(* write scene if necessary *)
IF swrite THEN
	status := 176;		(* write scene *)
	sx[x,0] := pi;
	sx[x,1] := ai;
	IF enable THEN sx[x,2] := 1; ELSE sx[x,2] := 0; END_IF; (* if sx[x,2] = 0 the scene is disabled *)
END_IF;


(* revision history
hm	24. oct 2007	rev 1.0
	original release

hm		29.1.2008	rev 1.1
	replaced shr/shl with and for better performance
*)
END_FUNCTION_BLOCK

(* POU BLIND_SECURITY, ST *)
FUNCTION_BLOCK BLIND_SECURITY
VAR_INPUT
	UP, DN : BOOL;
	S_IN : BYTE;
	pi, ai : BYTE;
	FIRE : BOOL;
	Wind : BOOL;
	Alarm : BOOL;
	Door : BOOL;
	Rain : BOOL;
END_VAR
VAR_INPUT CONSTANT
	Alarm_UP : BOOL := TRUE;
	WIND_UP :BOOL := TRUE;
	RAIN_UP : BOOL := FALSE;
END_VAR
VAR_OUTPUT
	QU, QD : BOOL;
	status : BYTE;
	po, ao : BYTE;
END_VAR
VAR
END_VAR

(*
version 1.2	12. feb 2008
programmer 	hugo
tested by		tobias


*)
IF Fire THEN
	QU := TRUE;
	QD := FALSE;
	status := 111;
ELSIF Wind THEN
	QU := Wind_up;
	QD := NOT wind_up;
	status := 112;
ELSIF alarm THEN
	QU := Alarm_up;
	QD := NOT Alarm_up;
	status := 113;
ELSIF Door THEN
	QU := TRUE;
	QD := FALSE;
	status := 114;
ELSIF Rain AND NOT (up XOR dn) THEN
	QU := rain_up;
	QD := NOT rain_up;
	status := 115;
ELSE
	QU := UP;
	QD := DN;
	status := S_IN;
	po := pi;
	ao := ai;
END_IF;


(* revision history
hm	29. sep 2007	rev 1.0
	original release

hm	6. oct 2007		rev 1.1
	added pos and angle inputs and outputs
	manual will override rain position
	alarm position can now be configured

hm		12. feb. 2008	rev 1.2
	added config variables rain_up and wind_up
	position for rain and wind is now configurable
*)
END_FUNCTION_BLOCK

(* POU BLIND_SHADE, ST *)
FUNCTION_BLOCK BLIND_SHADE
VAR_INPUT
	UP, DN : BOOL;
	S_IN : BYTE;
	pi, ai : BYTE;
	enable : BOOL;
	sun : BOOL;
	dtin : DT;
	sunrise, sunset : TOD;
	sun_hor, sun_ver : REAL;
END_VAR
VAR_INPUT CONSTANT
	sunrise_offset : TIME := T#1h;
	sunset_preset : TIME := T#1h;
	direction : REAL := 180;
	angle_offset : REAL := 80;
	slat_width : REAL := 80;
	Slat_spacing : REAL := 60;
	Shade_delay : TIME := T#60s;
END_VAR
VAR_OUTPUT
	QU, QD : BOOL;
	status : BYTE;
	po, ao : BYTE;
END_VAR
VAR
	angle: REAL;
	sun_delay : TOF;
END_VAR

(*
version 1.2	24 nov 2007
programmer 	hugo
tested by		tobias


*)
(* the input sun is sent through tof which will delay the shade for the time shade_delay *)
sun_delay(IN := sun, PT := shade_delay);

IF UP AND DN AND enable AND sun_delay.Q AND sun_hor > direction - angle_offset AND sun_hor < direction + angle_offset AND
	DT_TO_TOD(dtin) > sunrise + sunrise_offset AND DT_TO_TOD(dtin) < sunset - sunset_preset THEN
	status := 151;
	QU := UP;
	QD := DN;
	(* position is fully down *)
	po := 0;
	(* shading is active now calculate the slat angle *)
	(* calculate the max angle for the blind *)
	angle := DEG(ATAN(slat_spacing / slat_width));
	(* check if sun angle is between 0 and max angle *)
	IF sun_ver > 0 AND sun_ver < angle THEN
		angle := sun_ver + DEG(ACOS(COS(RAD(sun_ver))*slat_spacing / Slat_width));
		ao := INT_TO_BYTE(LIMIT(0,TRUNC(angle * 255 / 90), 255));
	ELSE
		ao := 255;
	END_IF;
ELSE
	QU := UP;
	QD := DN;
	po := pi;
	ao := ai;
	status := S_IN;
END_IF;

(* revision history
hm	15 oct. 2007	rev 1.0
	original version

hm	19. oct 2007	rev 1.1
	manual mode was not detected because outputs were checked and not inputs UP and DN

hm	24. nov 2007	rev 1.2
	added shade_delay to avoid constant up and down if sun is out parcially
*)
END_FUNCTION_BLOCK

(* POU DEG, ST *)
FUNCTION DEG : REAL
VAR_INPUT
	rad : REAL;
END_VAR
VAR
END_VAR
VAR
END_VAR

(*
version 1.1	16 oct 2007
programmer 	hugo
tested by		tobias

this function converts degrees into Radiant
execution time on wago 750 - 841 =  10  us
*)
deg := modR(57.29577951308232 * Rad, 360);

(* revision history
hm	4. aug 2006		rev 1.0
	original version

hm 	16. oct 2007	rev 1.1
	added modr statement which prohibits deg to become bigger than 360

*)
END_FUNCTION

(* POU RAD, ST *)
FUNCTION RAD : REAL
VAR_INPUT
	deg : REAL;
END_VAR
VAR
END_VAR

(*
version 1.0	4 aug 2006
programmer 	hugo
tested by	tobias

this function converts Radiant to degrees

*)
Rad := modR(0.0174532925199433 * deg,PI2);

(* revision history
hm	4. aug 2006
	original version

hm 	16. oct 2007
	added modr statement which prohibits rad to become bigger than 2PI

*)
END_FUNCTION

(* POU MODR, ST *)
FUNCTION MODR : REAL
VAR_INPUT
	in : REAL;
	divi : REAL;
END_VAR

VAR
END_VAR

(*
version 1.3	4. apr. 2008
programmer 	hugo
tested by	tobias

this is a modulo funtion for real numbers
modr(5.5,2.5) = 0.5

*)
IF divi = 0 THEN
	MODR := 0;
ELSE
	MODR := in - DINT_TO_REAL(D_TRUNC(in / divi)) * divi;
END_IF;

(* revision history

hm	4. aug.2006		rev 1.0

hm	28. jan.2007	rev 1.1
	modr(x,0) will deliver the result 0

hm	21. mar 2008	rev 1.2
	use D_trunc for compatibility reasons

hm	4. apr. 2008	rev 1.3
	added type conversion to avoid warnings under codesys 3.0

*)
END_FUNCTION

(* POU BOILER, ST *)
FUNCTION_BLOCK BOILER
VAR_INPUT
	T_upper : REAL;
	T_lower : REAL;
	Pressure : BOOL := TRUE;
	enable : BOOL := TRUE;
	Req_1 : BOOL;
	Req_2 : BOOL;
	Boost : BOOL;
END_VAR
VAR_INPUT CONSTANT
	t_upper_min : REAL := 50;
	t_upper_max : REAL := 60;
	T_lower_enable : BOOL;
	T_lower_max : REAL := 60;
	T_request_1 : REAL := 70;
	T_request_2 : REAL := 50;
	T_request_hys : REAL := 5;
	T_protect_high : REAL := 80;
	T_protect_low : REAL := 10;
END_VAR
VAR_OUTPUT
	Heat : BOOL;
	error : BOOL;
	status : BYTE;
END_VAR
VAR
	edge: BOOL;
	boost_mode: BOOL;
	flag_0 : BOOL;
	flag_1: BOOL;
	flag_2: BOOL;
END_VAR

(*
version 1.0	27 feb 2007
programmer 	hugo
tested by		tobias

this function block controls a hot water boiler. The Boiler can be equipped with two temperature sensors on top and bottom of the tank, T_LOWER_ENABLE must be set to True in this case.
alternatively can BOILER be configured for one (TOP) temperature sensor only (T_LOWER_ENABLE set to False).
A Pressure sensor is used to detect fresh water pressure and disable all heating if there is no water pressure. This input is dset to True by default, so if it is not used it can simply be left open.
A enable input enables the hot water heating while it is set to True. alternatively can a Ture on Req_1 or Req_2 start the heating to predefined temperatures during setup.
A low to high edge on the boost input will start heating imediately until T_upper_max is reached, it can be used to generate extra hot water when needed.

*)
(* read sensors and check for valid data *)
IF t_upper > t_protect_high THEN
	status := 1;
	heat := FALSE;
	error := TRUE;
ELSIF t_upper < t_protect_low THEN
	status := 2;
	heat := TRUE;
	error := TRUE;
ELSIF t_lower > T_protect_high AND t_lower_enable THEN
	status := 3;
	heat := FALSE;
	error := TRUE;
ELSIF t_lower < t_protect_low AND t_lower_enable THEN
	status := 4;
	heat := TRUE;
	error := TRUE;
ELSIF NOT pressure THEN
	status := 5;
	heat := FALSE;
	error := TRUE;
ELSIF req_1 OR req_2 OR enable OR boost THEN
	error := FALSE;

	(* determine if heat needs to be turned on *)
	IF boost AND NOT edge AND t_upper < t_upper_max THEN
		status := 101;
		heat := TRUE;
		boost_mode := TRUE;
	ELSIF enable AND t_upper < T_upper_min THEN
		status := 102;
		heat := TRUE;
	ELSIF req_1 AND t_upper < T_request_1 THEN
		status := 103;
		heat := TRUE;
	ELSIF req_2 AND t_upper < t_request_2 THEN
		status := 104;
		heat := TRUE;
	END_IF;

	(* determine the shut off temperature *)
	IF heat THEN
		IF (enable OR boost_mode) THEN
			flag_0 := TRUE;
			IF T_lower_enable AND T_lower > T_lower_max THEN
				flag_0 := FALSE;
				boost_mode := FALSE;
			ELSIF NOT T_lower_enable AND T_upper > T_upper_max THEN
				flag_0 := FALSE;
				boost_mode := FALSE;
			END_IF;
		ELSE
			flag_0 := FALSE;
		END_IF;
		IF req_1 AND T_upper > T_request_1 + T_request_hys THEN flag_1 := FALSE; ELSE flag_1 := req_1; END_IF;
		IF req_2 AND T_upper > T_request_2 + T_request_hys THEN flag_2 := FALSE; ELSE flag_2 := req_2; END_IF;

		(* shut off heat if no longer needed *)
		heat := flag_0 OR flag_1 OR flag_2;
		IF heat = FALSE THEN status := 100; END_IF;
	END_IF;
ELSE
	status := 100;
	heat := FALSE;
	error := FALSE;
END_IF;
edge := boost;
END_FUNCTION_BLOCK

(* POU PRESSURE, ST *)
FUNCTION_BLOCK PRESSURE
VAR_INPUT
	mws : REAL;
	torr : REAL;
	att : REAL;
	atm : REAL;
	pa : REAL;
	bar : REAL;
END_VAR
VAR_OUTPUT
	Ymws : REAL;
	Ytorr : REAL;
	Yatt : REAL;
	Yatm : REAL;
	Ypa : REAL;
	Ybar : REAL;
END_VAR
VAR
END_VAR

(*
version 1.0	27 mar 2007
programmer 	hugo
tested by		oscat

this function converts different pressure units
any unused input can simply be left open.
different inputs connected at the same time will be added up.
*)
Ybar := bar +
		pa / 100000 +
		0.980665 * att +
		1.01325 * atm +
		0.001333224 * torr +
		0.0980665 * mws;
Ymws := ybar / 0.0980665;
Ytorr := ybar / 0.001333224;
Yatt := ybar / 0.980665;
yatm := ybar / 1.01325;
Ypa := ybar * 100000;


(*
Druck, Pascal Pa 1 Pa = 1 N/m2 = 1 kg/(s2 �E m) . 0,75 �E 10.2 mmHg
mechanische 1 MPa = 1 N/mm2 . fur Festigkeitsangaben
Spannung Bar bar 1 bar = 105 Pa = 103 mbar = 105 kg/(s2 �E m)
Millimeter- mmHg 1 mmHg = 133,322 Pa = 1,333 22 mbar
Quecksilbersaule . nur in Heilkunde zulassig
physik. Atmosphare atm 1 atm = 1,013 25 bar
techn. Atmosphare at 1 at = 1 kp/cm2 = 0,980665 bar
Torr Torr 1 Torr = (101325/760) Pa = 1,333224 mbar
Meter-Wassersaule mWS 1 mWS = 9806,65 Pa = 98,0665 mbar
psi lbf/in2 1 lbf/in2 = 68,947 57 mbar = 6894,757 Pa

*)
END_FUNCTION_BLOCK

(* POU BUFFER_SEARCH, ST *)
FUNCTION BUFFER_SEARCH : INT
VAR_INPUT
	pt : POINTER TO ARRAY[0..32767] OF BYTE;
	size : UINT;
	str : STRING(STRING_LENGTH);
	pos : INT;
	ign : BYTE;
END_VAR
VAR
	ps : POINTER TO ARRAY[0..255] OF BYTE;
	i: INT;
	end: INT;
	k: INT;
	lx: INT;
END_VAR


(*
version 1.2	13. may. 2008
programmer 	hugo
tested by		tobias

this function will search for a string STR in an array of byte starting at position pos.
the function needs to be called:	buffer_search(adr("array"),sizeof("array"), STR, POS, IGN);
because this function works with pointers its very time efficient and it needs no extra memory.
The function returns the position of the first character of the string in the array if found.
a 0 is returned if the string is not found in the array.
The parameter IGN specifies a wildcard character in the search string.

*)
ps := ADR(str);
lx := LEN(str);
end := UINT_TO_INT(size) - lx;
lx := lx - 1;
FOR i := pos TO end DO
	FOR k := 0 TO lx DO
		IF (ps^[k] <> ign) AND (ps^[k] <> pt^[i+k]) THEN EXIT; END_IF;
	END_FOR;
	IF k > lx THEN
		BUFFER_SEARCH := i;
		RETURN;
	END_IF;
END_FOR;
BUFFER_SEARCH := 0;


(* revision History

hm 5. mar. 2008	rev 1.0
	original version

hm	16. mar. 2008	rev 1.1
	chaged type of input size to uint

hm	13. may. 2008	rev 1.2
	changed type of pointer to array[1..32767]
	changed size of string to STRING_LENGTH
*)
END_FUNCTION

(* POU BUFFER_TO_STRING, ST *)
FUNCTION BUFFER_TO_STRING : STRING(STRING_LENGTH)
VAR_INPUT
	pt : POINTER TO ARRAY[0..32767] OF BYTE;
	size : UINT;
	start : UINT;
	stop : UINT;
END_VAR
VAR
	ps : POINTER TO BYTE;
	i : INT;
END_VAR


(*
version 1.3	12. jun. 2008
programmer 	hugo
tested by		tobias

this function will retrieve a string from an array of byte starting at position start and stop at position stop.
the function needs to be called:	buffer_TO_String(adr("array"),sizeof("array"), start, stop);
because this function works with pointers its very time efficient and it needs no extra memory.

*)
ps := ADR(BUFFER_TO_STRING);
start :=MIN(start, size);
stop := MIN(stop, size);
(* check for maximum string_length *)
IF UINT_TO_INT(stop - start + 1) >= STRING_LENGTH THEN
	stop := start + INT_TO_UINT(string_length) - 1;
END_IF;

FOR i := UINT_TO_INT(start) TO UINT_TO_INT(stop) DO
	ps^ := pt^[i];
	ps := ps + 1;
END_FOR;

(* terminate the string *)
ps^ := 0;

(* revision History
hm 	5. mar. 2008	rev 1.0
	original version

hm	16. mar. 2008	rev 1.1
	changed type of input size to uint

hm	13. may. 2008	rev 1.2
	changed type of pointer to array[0..32767]
	changed size of string to STRING_LENGTH

hm	12. jun. 2008	rev 1.3
	check for pointer overrun
	change input start and stop to uint
	added type conversions to avoid warnings under codesys 3.0
*)
END_FUNCTION

(* POU BURNER, ST *)
FUNCTION_BLOCK BURNER
VAR_INPUT
	in : BOOL;
	stage2 : BOOL;
	over_temp : BOOL;
	oil_temp : BOOL := TRUE;
	Flame : BOOL;
	rst : BOOL;
	rst_timer : BOOL;
END_VAR
VAR_INPUT CONSTANT
	pre_heat_time : TIME := t#5s;
	pre_vent_time : TIME := t#15s;
	pre_ignite_time : TIME := t#5s;
	post_ignite_time : TIME := t#25s;
	stage2_delay : TIME := t#10s;
	safety_time : TIME := t#5s;
	lockout_time : TIME := t#10s;
	multiple_ignition : BOOL := TRUE;
	KW1 : REAL;
	KW2 : REAL;
END_VAR
VAR_OUTPUT
	motor : BOOL;
	coil1 : BOOL;
	coil2 : BOOL;
	pre_heat: BOOL;
	ignite : BOOL;
	runtime1 : REAL;
	runtime2 : REAL;
	KWh : REAL;
	cycles : REAL;
	status : BYTE;
	fail : BOOL;
END_VAR
VAR
	state : BYTE;
	last : TIME;
	tx: TIME;
	last_change: TIME;
	timer1 : ontime;
	timer2 : ontime;
	oil_temp_last: BOOL;
END_VAR

(*
version 1.5	15 sep 2007
programmer 	oscat
tested by		tobias

burner ist eine Oel-Brenner_steuerung fuer nichtmodulierende Oelbrenner
die steuerung kann ueber setup werte programmiert werden und entsprechenden brennern angepasst werden.
die vorheizzeit ist die zeit die eine oelvorwaermung aufgeheizt wird bevor der motor gestartet wird.
der eingang oil_temp gibt an ob die oil_temp erreicht wurde, er ist default auf true und kann auch offen gelassen werden.
die vorbelueftungszeit ist die zeit die der luefter laeuft bevor die oelzufuhr freigegeben wird.
die vorzuendzeit iust diejenige zeit die die zuendung vor offnen des oelventiel gestartet wird.
nachzuendzeit ist die zeit die nach entzuendung der flamme noch gezuendet wird.
die sicherheitszeit ist die zeit nach der die oelzufuhr gesperrt wird wenn keine flamme entsteht.
nach ablauf der sicherheitszeit wird ein fehler flag gesetzt und kann erst nach der sperrzeit wieder durch einen reset geloescht werden.
waehrend der sperrzeit ist keine weitere zuendung oder einschalten moeglich.
das flag mehrfachzuendung gibt an ob eine erloschene flamme in betrieb automatisch wieder gezuendet werden soll.
der flammwaechster liegt auf eingang flamme, ein uebertemperaturschutz auf dem eingang over_temp
der betriebsstundenzaehler gibt die brennerstunden in stunden als real ausgabewer an.
der ausgang motor steuert den luefter / pumpenmotor, oil_ventil schaltet das oil ventil und zuendung schaltet die zuendung ein.

if output fail > 0 an error happened and the output has an error code:
0 :	no error
1 :	pre heating time expired and oil temp input is not true
2 :	flame monitor is active during preheating time
3 :	flame monitor active during pre_ventilation_time
4 :	no ignoition during safety time
5 :	no flame during operation
9 :	overtemp input is true

*)
(* read system time *)
tx := DWORD_TO_TIME(T_PLC_MS());

(* check rst input and overtemp *)
IF rst OR over_temp OR state = 0 THEN
	IF status > 0 AND tx - last_change >= lockout_time AND rst THEN
		status := 110;
		fail := FALSE;
		state := 1;
	ELSE
		(* normaler reset *)
		motor := FALSE;
		coil1 := FALSE;
		coil2 := FALSE;
		ignite := FALSE;
		pre_heat := FALSE;
		IF over_temp THEN
			status := 9;
			fail := TRUE;
		END_IF;
		last_change := tx;
		last := tx;
		state := 1;
	END_IF;
END_IF;

(* check for timer rst and rst timer if true *)
IF rst_timer THEN
	timer1( rst := TRUE);
	timer1.rst := FALSE;
	timer2(rst := TRUE);
	timer2.rst := FALSE;
END_IF;

(* quit here if an error is present *)
IF (status > 0 AND status < 100) OR rst THEN RETURN; END_IF;

(* start sequence *)
CASE state OF

1:	(* in signal starts oil pre heating *)
	IF in AND flame THEN
		state := 7;
		pre_heat := FALSE;
		status := 2;
		last_change := tx;
	ELSIF in THEN
		pre_heat := TRUE;
		state := 2;
		last_change := tx;
	END_IF;

2:	(* after pre_heating time start motor *)
	IF (tx- last_change >= pre_heat_time AND oil_temp) OR (oil_temp AND NOT oil_temp_last) THEN
		motor := TRUE;
		state := 3;
		last_change := tx;
	(* pre_heat_time ist abgelaufen und oil_temp ist nicht aktiv *)
	ELSIF tx - last_change >= pre_heat_time AND NOT oil_temp THEN
		state := 7;
		pre_heat := FALSE;
		status := 1;
		last_change := tx;
	(* flame monitor cannot be active at this time *)
	ELSIF flame THEN
		state := 7;
		pre_heat := FALSE;
		status := 2;
		last_change := tx;
	END_IF;

3:	(* abwarten bis zündung eingeschaltet werden kann *)
	IF tx - last_change >= pre_vent_time - pre_ignite_time THEN
		ignite := TRUE;
		state := 4;
		last_change := tx;
	(* flame monitor cannot be active at this time *)
	ELSIF flame THEN
		state := 7;
		pre_heat := FALSE;
		motor := FALSE;
		status := 3;
		last_change := tx;
	END_IF;

4:	(* warten bis oelzufuhr geoeffnet werden darf *)
	IF tx - last_change >= pre_ignite_time THEN
		coil1 := TRUE;
		state := 5;
		last_change := tx;
	END_IF;

5:	(* warten auf flammwaechter und falls noetig abschalten *)
	IF tx - last_change >= safety_time OR flame THEN
		IF NOT flame THEN
			(* notabschaltung da flammwaechster nicht angesprochen hat *)
			state := 7;
			motor := FALSE;
			coil1 := FALSE;
			pre_heat := FALSE;
			ignite := FALSE;
			status := 4;
			last_change := tx;
		ELSE
			state := 6;
			last_change := tx;
		END_IF;
	END_IF;

6:	(* brenner läuft, flammueberwachung und nach ablauf der nachigniteszeit ignite abschalten *)
	IF NOT flame AND NOT multiple_ignition THEN
		(* notabschaltung da flammwaechster keine flamme meldet *)
		state := 7;
		motor := FALSE;
		coil1 := FALSE;
		coil2 := FALSE;
		pre_heat := FALSE;
		ignite := FALSE;
		status := 5;
		last_change := tx;
	ELSIF NOT flame AND multiple_ignition THEN
		ignite := TRUE;
		state := 5;
		coil2 := FALSE;
		last_change := tx;
	ELSE
		IF tx - last_change >= post_ignite_time THEN
			(* post_ignite_time abgelaufen, ignite abschalten *)
			ignite := FALSE;
		END_IF;
		IF tx - last_change >= stage2_delay AND stage2 THEN
			coil2 := TRUE;
		ELSE
			coil2 := FALSE;
		END_IF;
	END_IF;
END_CASE;

(* abschaltung wenn kein eingangssignal *)
IF NOT in THEN
	state := 1;
	motor := FALSE;
	coil1 := FALSE;
	coil2 := FALSE;
	ignite := FALSE;
	pre_heat := FALSE;
	last_change := tx;
END_IF;

(* runtimezähler *)
timer1(in := flame AND in AND motor AND coil1 AND NOT coil2);
timer2(in := flame AND in AND motor AND coil1 AND coil2);
runtime1 := timer1.ontime;
runtime2 := timer2.ontime;
cycles := timer1.cycles;
KWH := runtime1 * KW1 + runtime2 * KW2;

(* zeit fuer naechsten aufruf merken *)
last := tx;

(* set fail output IF ERROR and Status  if normal operation *)

IF status > 0 AND status < 100 THEN
	fail := TRUE;
ELSE
	fail := FALSE;
	IF NOT in THEN
		status := 110;
	ELSIF flame AND in AND motor AND coil2 AND coil1 THEN
		status := 113;
	ELSIF flame AND in AND motor AND coil1 THEN
		status := 112;
	ELSE
		status := 111;
	END_IF;
END_IF;


(*
31.12.2006	hm		rev 1.1
	added pre_heat timing and output
	flame monitor before ignition will generate error on status output
	added output for KWh

31.12.2006	hm		rev 1.2
	added oil_temp_input

31.12.2006	hm		rev 1.3
	changed status output to be byte instead of bool

22.1.2007		hm		rev 1.4
	renamed fail output to status
	added output cycles
	corrected an error while pre_heat would be on when an error was present
	added coil2 output and stage2 input

15.9.2007		hm		rev 1.5
	replaced Time() with T_PLC_MS for compatibility and performance reasons

*)
END_FUNCTION_BLOCK

(* POU BYTE_OF_BIT, ST *)
FUNCTION BYTE_OF_BIT : BYTE
VAR_INPUT
	B0:BOOL;
	B1:BOOL;
	B2:BOOL;
	B3:BOOL;
	B4:BOOL;
	B5:BOOL;
	B6:BOOL;
	B7:BOOL;
END_VAR
VAR
END_VAR

(*
version 1.1	 18. feb 2006
programmer 	hugo
tested by		tobias

this function creates a byte from 8 individual bits

*)
Byte_of_bit := SHL(SHL(SHL(SHL(SHL(SHL(SHL(BOOL_TO_BYTE(B7),1) OR BOOL_TO_BYTE(B6),1) OR BOOL_TO_BYTE(B5),1) OR BOOL_TO_BYTE(B4),1)
	OR BOOL_TO_BYTE(B3),1) OR BOOL_TO_BYTE(B2),1) OR BOOL_TO_BYTE(B1),1) OR BOOL_TO_BYTE(B0);


(* revision history

hm	4. aug 2006		rev 1.0
	original version

hm	18. feb. 2008	rev 1.1
	improved performance

*)
END_FUNCTION

(* POU BYTE_OF_DWORD, ST *)
FUNCTION BYTE_OF_DWORD : BYTE
VAR_INPUT
	in : DWORD;
	N : BYTE;
END_VAR
VAR
END_VAR

(*
version 1.1	2 jan 2008
programmer 	hugo
tested by		tobias

this function extracts a single byte from the nth position from right (right is lowest byte) 
the lower byte (starting with Bit0 from in) is selected with N=0.
*)
Byte_of_Dword := DWORD_TO_BYTE(SHR(in,n*8));

(* revision history
hm	17. jan 2007	rev 1.0
	original version

hm	2. jan 2008		rev 1.1
	improved performance

*)
END_FUNCTION

(* POU BYTE_TO_BITS, ST *)
FUNCTION_BLOCK BYTE_TO_BITS
VAR_INPUT
	IN: BYTE;
END_VAR
VAR_OUTPUT
	B0: BOOL;
	B1: BOOL;
	B2: BOOL;
	B3: BOOL;
	B4: BOOL;
	B5: BOOL;
	B6: BOOL;
	B7: BOOL;
END_VAR
VAR
END_VAR

(*
version 1.1	16. mar. 2008
programmer 	hugo
tested by		tobias

this Function Block extracts the 8 Bits from a byte


*)
B0 := IN.0;
B1 := IN.1;
B2 := IN.2;
B3 := IN.3;
B4 := IN.4;
B5 := IN.5;
B6 := IN.6;
B7 := IN.7;

(* revision history
hm		4. aug 2006	rev 1.0
	original version

hm		16. mar 2008	rev 1.1
	renamed from byte_to_bit to byte_to_bits for compatibility reasons

*)
END_FUNCTION_BLOCK

(* POU BYTE_TO_RANGE, ST *)
FUNCTION BYTE_TO_RANGE : REAL
VAR_INPUT
	X : BYTE;
	low : REAL;
	high : REAL;
END_VAR
VAR
END_VAR

(*
version 1.0	9. jan 2008
programmer 	hugo
tested by		tobias

Byte_to_Range converts a Byte into a real between low and high.

*)
Byte_to_Range := (high - low) * X / 255.0 + low;


(* revision history
hm	9. jan 2008		rev 1.0
	original version

*)
END_FUNCTION

(* POU BYTE_TO_STRB, ST *)
FUNCTION BYTE_TO_STRB : STRING(8)
VAR_INPUT
	IN : BYTE;
END_VAR
VAR
	i: INT;
	pt : POINTER TO BYTE;
END_VAR

(*
version 1.3	20. jun. 2008
programmer 	hugo
tested by	oscat

BYTE_TO_STRINGB converts a Byte to a String of Bits represented by '0' and '1' s.
The lowest order bit will be on the right and the high order bit on the left.

*)
(* pointer für die ausgabe ermitteln *)
pt := ADR(BYTE_TO_STRB);
(* die 8 ausgabecharacter ermitteln und schreiben *)
FOR i := 1 TO 8 DO
	pt^ := BOOL_TO_BYTE(in.7) + 48;
	in := SHL(in,1);
	pt := pt + 1;
END_FOR;

(* der ausgabestring muss noch mit 0 abgeschlossen werden *)
pt^ := 0;

(* code before rev 1.1
FOR i := 1 TO 8 DO
	IF in.0 = 0 THEN temp := CONCAT('0', temp); ELSE temp := CONCAT('1', temp); END_IF;
	in := SHR(in, 1);
END_FOR;
BYTE_TO_STRB := temp;
*)


(* revision history

hm		9.6.2007	rev 1.0		
	original version 

hm	15. dec 2007	rev 1.1
	inprooved code for higher performance

hm	29. mar. 2008	rev 1.2
	changed STRING to STRING(8)

hm	20. jun. 2008	rev 1.3
	performance improvement

*)
END_FUNCTION

(* POU BYTE_TO_STRH, ST *)
FUNCTION BYTE_TO_STRH : STRING(2)
VAR_INPUT
	IN : BYTE;
END_VAR
VAR
	temp : BYTE;
	PT : POINTER TO BYTE;
END_VAR

(*
version 1.3	29 mar. 2008
programmer 	hugo
tested by		tobias

BYTE_TO_STRINGH converts a Byte to a String of Hexadecimal represented by '0' .. '9' and 'A' .. 'F'.
The lowest order Character will be on the right and the high order Character on the left.

*)
(* read pointer to output string *)
PT := ADR(BYTE_TO_STRH);
(* calculate high order hex value *)
temp := SHR(in,4);
(* convert value to hex character *)
IF temp <= 9 THEN temp := temp + 48; ELSE temp := temp + 55; END_IF;
(* write friat character to output string *)
PT^ := temp;
(* calculate low order hex value *)
temp := in AND 2#00001111;
IF temp <= 9 THEN temp := temp + 48; ELSE temp := temp + 55; END_IF;
(* increment pointer and wirte low order character *)
pt := pt + 1;
pt^ := temp;
(* set pointer at the end of the output string and close the string with 0 *)
pt := pt + 1;
pt^:= 0;


(* code before rev 1.2
FOR i := 1 TO 2 DO
	X := in AND 2#1111;
	IF X <= 9 THEN X := X + 48; ELSE X := X + 55; END_IF;
	Cx := CHR(X);
	temp := CONCAT(Cx, temp);
	in := SHR(in,4);
END_FOR;
BYTE_TO_STRH := temp;
*)

(* revision history

hm	9.6.2007		rev 1.0		
	original version 

hm	11.9.2007		rev 1.1		
	changed coding for compatibility with twincat, under twincat concat cannot have a function as argument.	

hm	15 dec 2007		REV 1.2
	changed code for higher performance

hm	29. mar. 2008	rev 1.3
	changed STRING to STRING(2)
*)
END_FUNCTION

(* POU C_TO_F, ST *)
FUNCTION C_TO_F : REAL
VAR_INPUT
	celsius : REAL;
END_VAR
VAR
END_VAR

(*
version 1.0	4 aug 2006
programmer 	hugo
tested by		tobias

this function converts celsius  to fahrenheit 

*)
C_to_F := celsius * 1.8 + 32;
END_FUNCTION

(* POU C_TO_K, ST *)
FUNCTION C_TO_K : REAL
VAR_INPUT
	Celsius : REAL;
END_VAR
VAR
END_VAR

(*
version 1.0	4 dec 2006
programmer 	hugo
tested by		tobias

this function converts celsius to kelvin
*)
C_to_K := Celsius - 273.15;
END_FUNCTION

(* POU CABS, ST *)
FUNCTION CABS : REAL
VAR_INPUT
	X : complex;
END_VAR
VAR
END_VAR

(*
version 1.0	21 feb 2008
programmer 	hugo
tested by	oscat

this function the aboslute value of a complex number

*)
CABS := HYPOT(x.re, x.im);


(* revision history
hm	21. feb 2008	rev 1.0
	original version

*)
END_FUNCTION

(* POU HYPOT, ST *)
FUNCTION HYPOT : REAL
VAR_INPUT
	X : REAL;
	Y : REAL;
END_VAR
VAR
END_VAR

(*
version 1.0	21 feb 2008
programmer 	hugo
tested by	oscat

this function calculates the pythagorean function

*)
HYPOT := SQRT(x*x + y*y);


(* revision history
hm	21. feb 2008	rev 1.0
	original version

*)
END_FUNCTION

(* POU CACOS, ST *)
FUNCTION CACOS : complex
VAR_INPUT
	X : complex;
END_VAR
VAR
	Y : complex;
END_VAR

(*
version 1.0	21 feb 2008
programmer 	hugo
tested by	oscat

this function calculates the arcus cosinus function of a complex number

*)
y := CACOSH(x);
CACOS.re := y.im;
CACOS.im := -y.re;



(* revision history
hm	21. feb 2008	rev 1.0
	original version


*)
END_FUNCTION

(* POU CACOSH, ST *)
FUNCTION CACOSH : complex
VAR_INPUT
	X : complex;
END_VAR
VAR
	Y : complex;
END_VAR

(*
version 1.0	21 feb 2008
programmer 	hugo
tested by	oscat

this function calculates the hyperbolic arcus cosinus function of a complex number

*)
y.re := (X.re - X.im)*(X.re + X.im) - 1.0;
y.im := 2.0 * X.re * X.im;
y    := CSQRT(y);
y.re := y.re + x.re;
y.im := y.im + x.im;
CACOSH  := CLOG(y);



(* revision history
hm	21. feb 2008	rev 1.0
	original version


*)
END_FUNCTION

(* POU CSQRT, ST *)
FUNCTION CSQRT : complex
VAR_INPUT
	X : complex;
END_VAR
VAR
	temp : REAL;
END_VAR

(*
version 1.0	21 feb 2008
programmer 	hugo
tested by	oscat

this function calculates the complex sqare root

*)
temp := HYPOT(x.re, x.im);
CSQRT.re :=  SQRT(0.5 * (temp + x.re));
CSQRT.im :=  sgn(x.im) * SQRT(0.5 * (temp - x.re));


(* revision history
hm	21. feb 2008	rev 1.0
	original version

*)
END_FUNCTION

(* POU SGN, ST *)
FUNCTION SGN : INT
VAR_INPUT
	X : REAL;
END_VAR
VAR
END_VAR

(*
version 1.1	11. nov. 2008
programmer 	hugo
tested by	tobias

sgn returns 0 when X = 0 , -1 when X < 1 and +1 when X > 1

*)
IF X > 0 THEN
	SGN := 1;
ELSIF X < 0 THEN
	SGN := -1;
ELSE
	SGN := 0;
END_IF;



(* revision histroy
hm	16. oct 2007	rev 1.0
	original version

hm	11. nov 2007	rev 1.1
	changed type of function from real to int

*)
END_FUNCTION

(* POU CLOG, ST *)
FUNCTION CLOG : complex
VAR_INPUT
	X : complex;
END_VAR
VAR
END_VAR

(*
version 1.1	20. apr. 2008
programmer 	hugo
tested by	oscat

this function calculates the complex natural (base e) logarithm

*)
CLOG.re := LN(HYPOT(X.re, X.im));
CLOG.im := ATAN2(X.im, X.re);


(* revision history
hm	21. feb 2008	rev 1.0
	original version

hm	20. apr. 2008	rev 1.1
	use ATAN2 instead of ATAN
*)
END_FUNCTION

(* POU CADD, ST *)
FUNCTION CADD : complex
VAR_INPUT
	X, Y : complex;
END_VAR
VAR
END_VAR

(*
version 1.0	21 feb 2008
programmer 	hugo
tested by	oscat

this function add two complex numbers

*)
CADD.re := x.re + y.re;
CADD.im := x.im + y.im;


(* revision history
hm	21. feb 2008	rev 1.0
	original version

*)
END_FUNCTION

(* POU CALIBRATE, ST *)
FUNCTION_BLOCK CALIBRATE
VAR_INPUT
	X : REAL;
	CO : BOOL;
	CS : BOOL;
END_VAR
VAR_INPUT CONSTANT
	Y_Offset : REAL;
	Y_Scale : REAL;
END_VAR
VAR_OUTPUT
	Y : REAL;
END_VAR
VAR RETAIN
	offset : REAL;
	Scale : REAL := 1;
END_VAR

(*
	version 1.2	22 feb 2007
	programmer 	hugo
	tested BY		hans

Calibrate allows for offset and scale calibration of an analog input.
offset is calibrated to a stored reference Y_offset while CO is true.
after the offset is calibrated, scale can be calibrated to a reference value Y_scale while CS is true.
*)
(* check for calibration *)
IF CO THEN
	Offset := Y_Offset - X;
ELSIF CS THEN
	scale := Y_scale / (X+Offset);
END_IF;
(* calculate output *)
Y := (X + Offset) * Scale;


(* revision history
hm 22.2.2007		rev 1.2
	changed VAR RETAIN PERSISTENT to VAR RETAIN for better compatibility
	wago lon contollers do not support persisitent

*)
END_FUNCTION_BLOCK

(* POU SCALE, ST *)
FUNCTION SCALE : REAL
VAR_INPUT
	X : REAL;
	K : REAL;
	O : REAL;
	MX : REAL;
	MN : REAL;
END_VAR
VAR
END_VAR

(*
version 1.0	16. may. 2008
programmer 	hugo
tested by		tobias

Scale is used to translate an input x to output by the formula Y = X*K + O.
at the same time the output is limited to MN and MX.

*)
SCALE := LIMIT(MN, X * K + O, MX);


(* revision history
hm	16. may. 2008		rev 1.0
	original version
*)
END_FUNCTION

(* POU CAPITALIZE, ST *)
FUNCTION CAPITALIZE : STRING(STRING_LENGTH)
VAR_INPUT
	str : STRING(STRING_LENGTH);
END_VAR
VAR
	PT : POINTER TO BYTE;
	pos : INT;
	L : INT;
	first : BOOL := TRUE;
END_VAR

(*
version 1.2	20. jun. 2008
programmer 	hugo
tested by		tobias

uppercase returns str while all letters a..z and ä,ö,ü are converted to uppercase

*)
PT := ADR(CAPITALIZE);
CAPITALIZE := str;
L := LEN(str);
FOR pos := 1 TO l DO
	IF first THEN pt^ := TO_UPPER(pt^);	END_IF;
	(* remember in first if the next char needs to capitalized *)
	first := pt^= 32;
	PT := pt + 1;
END_FOR;

(* revision histroy
hm		4. mar 2008	rev 1.0
	original release

hm	29. mar. 2008	rev 1.1
	changed STRING to STRING(STRING_LENGTH)

hm	20. jun. 2008	rev 1.2
	improved performance

*)	
END_FUNCTION

(* POU TO_UPPER, ST *)
FUNCTION TO_UPPER : BYTE
VAR_INPUT
	IN : BYTE;
END_VAR
VAR
END_VAR

(*
version 1.0	6 mar 2008
programmer 	hugo
tested by		tobias

to_upper converts a character from lowercase to uppercase

*)
IF extended_ascii THEN
	IF ((in > 96) AND (in < 123)) OR ((in > 223) AND (in <> 247) AND (in <> 255)) THEN
		TO_UPPER := in AND 16#DF;
	ELSE
		TO_UPPER := in;
	END_IF;
ELSE
	IF ((in > 96) AND (in < 123)) THEN
		TO_UPPER := in AND 16#DF;
	ELSE
		TO_UPPER := in;
	END_IF;
END_IF;

(* revision history
hm		6. mar 2008	rev 1.0
	original version

*)
END_FUNCTION

(* POU CARG, ST *)
FUNCTION CARG : REAL
VAR_INPUT
	X : complex;
END_VAR
VAR
END_VAR

(*
version 1.1	20. apr. 2008
programmer 	hugo
tested by	oscat

this function calculates the phase angle (argument) of a complex number

*)
CARG := ATAN2(X.im, X.re);



(* revision history
hm	21. feb. 2008	rev 1.0
	original version

hm	20. apr. 2008	rev 1.1
	use ATAN2 instead of ATAN
*)
END_FUNCTION

(* POU CASIN, ST *)
FUNCTION CASIN : complex
VAR_INPUT
	X : complex;
END_VAR
VAR
	Y : complex;
END_VAR

(*
version 1.0	21 feb 2008
programmer 	hugo
tested by	oscat

this function calculates the arcus sinus function of a complex number

*)
y.re := -x.im;
y.im := x.re;
y := CASINH(y);
CASIN.re := y.im;
CASIN.im := -y.re;



(* revision history
hm	21. feb 2008	rev 1.0
	original version


*)
END_FUNCTION

(* POU CASINH, ST *)
FUNCTION CASINH : complex
VAR_INPUT
	X : complex;
END_VAR
VAR
	Y : complex;
END_VAR

(*
version 1.0	21 feb 2008
programmer 	hugo
tested by	oscat

this function calculates the hyperbolic arcus sinus function of a complex number

*)
y.re := (X.re - X.im)*(X.re + X.im) + 1.0;
y.im := 2.0 * X.re * X.im;
y    := CSQRT(y);
y.re := y.re + x.re;
y.im := y.im + x.im;
CASINH  := CLOG(y);



(* revision history
hm	21. feb 2008	rev 1.0
	original version


*)
END_FUNCTION

(* POU CATAN, ST *)
FUNCTION CATAN : complex
VAR_INPUT
	X : complex;
END_VAR
VAR
	r2: REAL;
	num, den : REAL;
END_VAR

(*
version 1.0	21 feb 2008
programmer 	hugo
tested by	oscat

this function calculates the complex arcus tangens

*)
r2 := x.re * x.re;
den := 1.0 - r2 - x.im * x.im;
CATAN.re := 0.5 * ATAN(2.0 * x.re / den);
num := x.im + 1.0;
num := r2 + num * num;
den := x.im - 1.0;
den := r2 + den * den;
CATAN.im := 0.25 * (LN(num)-LN(den));

(* revision history
hm	21. feb 2008	rev 1.0
	original version


*)
END_FUNCTION

(* POU CATANH, ST *)
FUNCTION CATANH : complex
VAR_INPUT
	X : complex;
END_VAR
VAR
	i2: REAL;
	num, den : REAL;
END_VAR

(*
version 1.0	21 feb 2008
programmer 	hugo
tested by	oscat

this function calculates the complex arcus hyperbolic tangens

*)
i2 := x.im * x.im;
num := 1.0 + x.re;
num := i2 + num * num;
den := 1.0 - x.re;
den := i2 + den * den;
CATANH.re := 0.25 * (LN(num) - LN(den));
den := 1 - x.re * x.re - i2;
CATANH.im := 0.5 * ATAN(2.0 * x.im / den);

(* revision history
hm	21. feb 2008	rev 1.0
	original version


*)
END_FUNCTION

(* POU CCON, ST *)
FUNCTION CCON : complex
VAR_INPUT
	X : complex;
END_VAR
VAR
END_VAR

(*
version 1.0	21 feb 2008
programmer 	hugo
tested by	oscat

this function calcucates the conjugation of a complex number

*)
CCON.re := x.re;
CCON.im := -x.im;


(* revision history
hm	21. feb 2008	rev 1.0
	original version

*)
END_FUNCTION

(* POU CCOS, ST *)
FUNCTION CCOS : complex
VAR_INPUT
	X : complex;
END_VAR
VAR
END_VAR

(*
version 1.0	21 feb 2008
programmer 	hugo
tested by	oscat

this function calculates the cosinus function of a complex number

*)
CCOS := CCOSH(CSET(-X.im, X.re));


(* revision history
hm	21. feb 2008	rev 1.0
	original version

*)
END_FUNCTION

(* POU CCOSH, ST *)
FUNCTION CCOSH : complex
VAR_INPUT
	X : complex;
END_VAR
VAR
END_VAR

(*
version 1.0	21 feb 2008
programmer 	hugo
tested by	oscat

this function calculates the arcus tangens function of a complex number

*)
CCOSH.re := cosH(x.re) * COS(x.im);
CCOSH.im := sinH(x.re) * SIN(x.im);


(* revision history
hm	21. feb 2008	rev 1.0
	original version

*)
END_FUNCTION

(* POU COSH, ST *)
FUNCTION COSH : REAL
VAR_INPUT
	X : REAL;
END_VAR
VAR
	t: REAL;
END_VAR


(*
version 1.2	5. jan 2008
programmer 	hugo
tested by		tobias

this function calculates the cos hyperbolicus

*)
T := EXP(X);
COSH := (1/T + T) * 0.5;

(* revision histroy
hm	12.1.2007	rev 1.0
	original version

hm	1.12.2007	rev 1.1
	changed code to improve performance

hm	5. jan 2008	rev 1.2
	further performance improvement
*)
END_FUNCTION

(* POU SINH, ST *)
FUNCTION SINH : REAL
VAR_INPUT
	X : REAL;
END_VAR
VAR
END_VAR


(*
version 1.3	11. mar 2008
programmer 	hugo
tested by	tobias

this function calculates the sin hyperbolicus

*)
IF ABS(x) < 2E-3 THEN
	SINH := X;
ELSE
	SINH := (EXP(x) - EXP(-x)) * 0.5;
END_IF;


(* revision history
hm	12.1.2007	rev 1.0
	original version

hm	1.12.2007	rev 1.1
	changed code to improve performance

hm	5. jan 2008	rev 1.2
	further performance improvement

hm	11. mar 2008	rev 1.3
	improved accuracy around 0

*)
END_FUNCTION

(* POU CSET, ST *)
FUNCTION CSET : complex
VAR_INPUT
	RE : REAL;
	IM : REAL;
END_VAR
VAR
END_VAR

(*
version 1.0	21 feb 2008
programmer 	hugo
tested by	oscat

this function creates a complex number from two real inputs

*)
CSET.re := RE;
CSET.im := IM;

(* revision history
hm	21. feb 2008	rev 1.0
	original version

*)
END_FUNCTION

(* POU CDIV, ST *)
FUNCTION CDIV : complex
VAR_INPUT
	X, Y : complex;
END_VAR
VAR
	Temp : REAL;
END_VAR

(*
version 1.0	21 feb 2008
programmer 	hugo
tested by	oscat

this function divides two complex numbers

*)
temp := Y.re * Y.re + Y.im * Y.im;
CDIV.re := (X.re * Y.re + X.im * Y.im) / temp;
CDIV.im := (X.im * Y.re - X.re * Y.im) / temp;

(* revision history
hm	21. feb 2008	rev 1.0
	original version

*)
END_FUNCTION

(* POU CEIL, ST *)
FUNCTION CEIL : INT
VAR_INPUT
	X : REAL;
END_VAR
VAR
END_VAR


(*
version 1.1	21. mar. 2008
programmer 	hugo
tested by	tobias

This is a rounding function which returns the smallest possible integer which is greater or equal to X.
ceil(3.14) = 4
ceil(-3.14) = -3

*)
CEIL := REAL_TO_INT(x);
IF CEIL < X THEN
	CEIL := CEIL + 1;
END_IF;

(* code used for rev 1.0
CEIL := D_TRUNC(X);
IF CEIL < X THEN
	ceil := ceil + 1;
END_IF;
*)

(* revision history
hm	7. feb. 2007	rev 1.0
	original version

hm	21. mar. 2008	rev 1.1
	use REAL_TO_INT instead of trunc for compatibility reasons


*)
END_FUNCTION

(* POU CEIL2, ST *)
FUNCTION CEIL2 : DINT
VAR_INPUT
	X : REAL;
END_VAR
VAR
END_VAR


(*
version 1.2	30. jun. 2008
programmer 	hugo
tested by	tobias

This is a rounding function which returns the smallest possible integer which is greater or equal to X.
ceil2(3.14) = 4
ceil2(-3.14) = -3

*)
CEIL2 := REAL_TO_INT(X);
IF DINT_TO_REAL(CEIL2) < X THEN
	CEIL2 := CEIL2 + 1;
END_IF;


(* revision history
hm	21. mar. 2008	rev 1.0
	original version

hm	4. apr. 2008	rev 1.1
	added type conversion to avoid warnings under codesys 3.0

hm	30. jun. 2008	rev 1.2
	added type conversion to avoid warnings under codesys 3.0
*)
END_FUNCTION

(* POU CEXP, ST *)
FUNCTION CEXP : complex
VAR_INPUT
	X : complex;
END_VAR
VAR
	Temp : REAL;
END_VAR

(*
version 1.0	21 feb 2008
programmer 	hugo
tested by	oscat

this function calculates the complex exponent

*)
temp := EXP(X.re);
CEXP.re := temp * COS(X.im);
CEXP.im := temp * SIN(X.im);


(* revision history
hm	21. feb 2008	rev 1.0
	original version

*)
END_FUNCTION

(* POU CHARCODE, ST *)
FUNCTION CHARCODE : BYTE
VAR_INPUT
	STR : STRING(10);
END_VAR
VAR
	found: STRING(1);
	search : STRING(10);
	pos: INT;
END_VAR

(*
version 1.0		13. may. 2008
programmer 		hugo
tested by			hugo

CHARCODE converts a HTML Character NAME INTO ITS code
'äuml' is convterted to ä
'euro' is converted to €

*)
(* return 0 if empty string *)
IF str = '' THEN
	RETURN;
ELSIF STR = '&' THEN
	CHARCODE := 33;
	RETURN;
ELSIF str = ';' THEN
	CHARCODE := 59;
	RETURN;
END_IF;

(* construct search string *)
search := CONCAT('&', str);
search := CONCAT(search, ';');

(* search the 4 strings for ocurence and read preceding code if found*)
pos := FIND(CHARNAME_1, search);
IF pos > 0 THEN
	found := MID(CHARNAME_1, 1, pos - 1);
ELSE
	pos := FIND(CHARNAME_2, search);
	IF pos > 0 THEN
		found := MID(CHARNAME_2, 1, pos - 1);
	ELSE
		pos := FIND(CHARNAME_3, search);
		IF pos > 0 THEN
			found := MID(CHARNAME_3, 1, pos - 1);
		ELSE
			pos := FIND(charname_4, search);
			IF pos > 0 THEN found := MID(CHARNAME_4, 1, pos - 1); END_IF;
		END_IF;
	END_IF;
END_IF;

(* convert to code *)
IF pos > 0 THEN
	CHARCODE := CODE(found, 1);
ELSE
	CHARCODE := CODE(STR, 1);
END_IF;


(* revision history
hm		13. may. 2008	rev 1.0
	original version

*)
END_FUNCTION

(* POU CODE, ST *)
FUNCTION CODE : BYTE
VAR_INPUT
	STR : STRING(STRING_LENGTH);
	POS : INT;
END_VAR
VAR
	PT : POINTER TO BYTE;
END_VAR

(*
version 1.1	29. mar. 2008
programmer 	hugo
tested by		tobias

code extracts the code of a character at position POS of a string STR.

*)
IF pos < 1 OR pos > LEN(str) THEN
	CODE := 0;
	RETURN;
ELSE
	PT := ADR(STR) + INT_TO_DWORD(pos - 1);
	CODE := pt^;
END_IF;

(* revision history
hm	9. mar. 2008	rev 1.0
	original version

hm	29. mar. 2008	rev 1.1
	changed STRING to STRING(STRING_LENGTH)
*)
END_FUNCTION

(* POU CHARNAME, ST *)
FUNCTION CHARNAME : STRING(10)
VAR_INPUT
	C : BYTE;
END_VAR
VAR
	search: STRING;
	pos: INT;
END_VAR

(*
version 1.1		16. jun. 2008
programmer 		hugo
tested by		oscat

CHARNAME converts a Character code into its HTML character name
ä is convterted to 'äuml'
€ is converted to 'euro'
the character itself is returned if no name is available for the character

*)
CHARNAME := CHR(C);
(* return empty string if code is 0 *)
IF C = 0 THEN RETURN; END_IF;

(* construct search string from code followed by $ sign, also clear charname string*)
search := CHR(C);
search := CONCAT(search,'&');
search := CONCAT(';', search);

(* search the 4 strings for ocurence and copy the following 10 chars if found*)
pos := FIND(CHARNAME_1, search);
IF pos > 0 THEN
	CHARNAME := MID(CHARNAME_1, 10, pos + 3);
ELSE
	pos := FIND(CHARNAME_2, search);
	IF pos > 0 THEN
		CHARNAME := MID(CHARNAME_2, 10, pos + 3);
	ELSE;
		pos := FIND(CHARNAME_3, search);
		IF pos > 0 THEN
			CHARNAME := MID(CHARNAME_3, 10, pos + 3);
		ELSE
			pos := FIND(CHARNAME_4, search);
			IF pos > 0 THEN CHARNAME := MID(CHARNAME_4, 10, pos + 3); END_IF;
		END_IF;
	END_IF;
END_IF;

(* search for end of name and truncate *)
IF pos > 0 THEN
	pos := FIND(CHARNAME, ';');
	CHARNAME := LEFT(CHARNAME,pos - 1);
END_IF;


(* revision history
hm	13. may. 2008	rev 1.0
	original version

hm	16. jun. 2008	rev 1.1
*)
END_FUNCTION

(* POU CHR, ST *)
FUNCTION CHR : STRING(1)
VAR_INPUT
	C : BYTE;
END_VAR
VAR
	PT : POINTER TO BYTE;
END_VAR

(*
version 1.2	29. mar. 2008
programmer 	hugo
tested by		tobias

CHR creates a character from a byte input and stuffs it in a one character length string.

*)
PT := ADR(CHR);
PT^ := C;
pt := pt + 1;
pt^ := 0;

(* revision history
hm	16 jan 2007		rev 1.0
	original version

hm	4. feb. 2008	rev 1.1
	return string would not be terminated properly

hm	29. mar. 2008	rev 1.2
	changed STRING to STRING(1)
*)
END_FUNCTION

(* POU CHECK_PARITY, ST *)
FUNCTION CHECK_PARITY : BOOL
VAR_INPUT
	in : DWORD;
	p : BOOL;
END_VAR
VAR
END_VAR

(*
version 1.3	18 feb 2008
programmer 	hugo
tested by		tobias

this function checks for an even partity for a dword and partity bit.

*)
check_parity := NOT p;
WHILE in > 0 DO
	check_parity := check_parity XOR in.0 XOR in.1 XOR in.2 XOR in.3;
	in := SHR(in,4);
END_WHILE;

(* code before rev 1.2
WHILE in > 0 DO
	IF in.0 THEN cnt := cnt + 1; END_IF;
	in := SHR(in,1);
END_WHILE;
check_parity := even(cnt) XOR P;
*)


(* revision history

rev 1.0 HM  1.oct.2006

rev 1.1 hm	10.sep.2007
	changed algorithm to improove performance

rev 1.2	hm	8 dec 2007
	changed algorithm to improove performance

rev 1.3 hm	18. feb 2008
	changed algorithm to improove performance
*)
END_FUNCTION

(* POU CINV, ST *)
FUNCTION CINV : complex
VAR_INPUT
	X : complex;
END_VAR
VAR
	temp : REAL;
END_VAR

(*
version 1.0	21 feb 2008
programmer 	hugo
tested by	oscat

this function calculates the inverse of a complex numbers (1 / X)

*)
temp := X.re * X.re + X.im * X.im;
CINV.re := X.re / temp;
CINV.im := -X.im / temp;

(* revision history
hm	21. feb 2008	rev 1.0
	original version

*)
END_FUNCTION

(* POU CIRCLE_A, ST *)
FUNCTION CIRCLE_A : REAL
VAR_INPUT
	rx : REAL;
	ax : REAL;
END_VAR
VAR
END_VAR

(*
version 1.2	22. feb 2008
programmer 	hugo
tested by		tobias

circle_A calculates the Area of a circle segement if ax = 360 the whole circle is calculated


*)
circle_A := Rx * RX * 8.726646E-3 * Ax;

(* revision histroy
hm	16. oct 2007	rev 1.0
	original version

hm	4. dec 2007		rev 1.1
	changed code for better performance

hm	22. feb 2008	rev 1.2
	improved performance
*)
END_FUNCTION

(* POU CIRCLE_C, ST *)
FUNCTION CIRCLE_C : REAL
VAR_INPUT
	Rx : REAL;
	Ax : REAL;
END_VAR
VAR
END_VAR

(*
version 1.1	22 feb 2008
programmer 	hugo
tested by		tobias

circle_C calculates the Circumference of a circle  if ax = 360 the whole circle is calculated

*)
circle_C := 1.7453293E-2 * Rx * Ax;

(* revision histroy
hm	16. oct 2007	rev 1.0
	original version

hm	22. feb 2008	rev 1.1
	improved performance
*)
END_FUNCTION

(* POU CLEAN, ST *)
FUNCTION CLEAN : STRING(STRING_LENGTH)
VAR_INPUT
	IN : STRING(STRING_LENGTH);
	CX : STRING(80);
END_VAR
VAR
	pos: INT := 1;
	stop: INT;
END_VAR


(*
version 1.0	18. jun. 2008
programmer 	hugo
tested by	oscat

Clean deletes all characters from a string except the ones specified in CX.

*)
(* copy input string *)
CLEAN := IN;
stop := LEN(in);
WHILE pos <= stop DO
	IF FIND(cx, MID(CLEAN, 1, pos)) > 0 THEN
		(* charcter found skip to next one *)
		pos := pos + 1;
	ELSE
		(* wrong chracter needs to be deleted *)
		CLEAN := DELETE(CLEAN, 1, pos);
		stop := stop - 1;	(* the string is one character shorter now *)
	END_IF;
END_WHILE;



(* revision history

hm		18. jun. 2008	rev 1.0		
	original version 


*)
END_FUNCTION

(* POU CLICK, ST *)
FUNCTION_BLOCK CLICK
VAR_INPUT
	in : BOOL;
END_VAR
VAR_OUTPUT
	Q : BOOL;
	single : BOOL;
	double : BOOL;
	triple : BOOL;
	status: BYTE;
END_VAR
VAR_INPUT CONSTANT
	T_debounce : TIME := t#10ms;
	T_short : TIME := t#200ms;
	T_pause : TIME := t#500ms;
	T_reconfig : TIME := t#1m;
END_VAR
VAR
	debounce : TON;
	tx : TIME;
	last : TIME;
	init : BOOL;
	edge : BOOL;
	standby: BOOL;
	state: INT;
END_VAR

(*
version 1.2	15 sep 2007
programmer 	oscat
tested by		tobias

click checks an input for single, double or tripple click and sets the corresponding output single, doulbe or triple for the time the input stays high at the last click.
the maximum high and low time for a click can beconfigrured with setup variables.
the input cinfigures itself to be high or low active dependung on which state the input stays longer than t_reconfig.

*)
(* read system time *)
tx := DWORD_TO_TIME(T_PLC_MS());

(* set last and tx if never started before *)
IF NOT init THEN
	init := TRUE;
	last := tx;
	debounce.PT := T_debounce;
	standby := in;
END_IF;

(* debounce input *)
debounce(in := in XOR standby);
Q := debounce.Q;

(* delete outputs if input is inactive *)
IF NOT Q THEN
	single := FALSE;
	double := FALSE;
	triple := FALSE;
	status := 110;
END_IF;

(* check for input edge *)
IF Q XOR edge THEN
	edge := in;
	last := tx;
	IF Q THEN state := state + 1; END_IF;
END_IF;

IF (q AND tx - last >= T_short) OR (NOT q AND tx - last >= t_pause) THEN
	CASE state OF
		1:	single := TRUE;
			status := 111;
		2:	double := TRUE;
			status := 112;
		3:	triple := TRUE;
			status := 113;
	END_CASE;
	state := 0;
END_IF;

(* determine if high or low active *)
IF tx - last >= t_reconfig THEN
	standby := in;
	last := tx;
END_IF;



(* revision history

15 Feb 2007	rev 1.0	hm
	created original version

18.5.2007		rev 1.1 hm
	corrected an error while execution would stop after t_reconfig elapsed.

15.9.2007		rev 1.2 hm
	replaced Time() with T_PLC_MS for compatibility and performance reasons

*)
END_FUNCTION_BLOCK

(* POU CLK_DIV, ST *)
FUNCTION_BLOCK CLK_DIV
VAR_INPUT
	clk : BOOL;
	rst: BOOL;
END_VAR
VAR_OUTPUT
	Q0 : BOOL := 0;
	Q1 : BOOL := 0;
	Q2 : BOOL := 0;
	Q3 : BOOL := 0;
	Q4 : BOOL := 0;
	Q5 : BOOL := 0;
	Q6 : BOOL := 0;
	Q7 : BOOL := 0;
END_VAR
VAR
	cnt: BYTE := 0;
END_VAR

(*
version 1.1	2 jan 2008
programmer 	hugo
tested by		tobias

this is a clock divider
each output divides the signal by 2
Q0 = clk / 2 , Q1 = Q0 / 2 and so on.
the outputs have a 50% duty cycle each.


*)
IF rst THEN
	cnt:= 0;
	Q0 := 0;
	Q1 := 0;
	Q2 := 0;
	Q3 := 0;
	Q4 := 0;
	Q5 := 0;
	Q6 := 0;
	Q7 := 0;
ELSIF clk THEN
	cnt:= cnt +1;
	Q0 := cnt.0;
	Q1 := cnt.1;
	Q2 := cnt.2;
	Q3 := cnt.3;
	Q4 := cnt.4;
	Q5 := cnt.5;
	Q6 := cnt.6;
	Q7 := cnt.7;
END_IF;

(* revision history
hm	4. aug. 2006	rev 1.0
	original version

hm	2. jan 2008		rev 1.1
	improved performance

*)
END_FUNCTION_BLOCK

(* POU CLK_N, ST *)
FUNCTION_BLOCK CLK_N
VAR_INPUT
	N : INT;
END_VAR
VAR_OUTPUT
	Q : BOOL;
END_VAR
VAR
	edge : BOOL := 0;
	stime: DWORD;
	clk: BOOL;
END_VAR

(*
version 1.0	17 sep 2007
programmer 	hugo
tested by		tobias

clk_N uses the internal sps time to generate one pulse every N ms
every pulse is only valid for one cycle so that a edge trigger is not necessary
clk_N generates pulses depending on the accuracy of the system clock.
The input N controlls the period time of the clock.
N=0 equals 1ms, N=1 equals 2ms, N=2 equals 4ms, N=3 equals 8ms ....

be careful, 1ms clocks will only work on very powerful sps cpu's
*)
stime := SHR(T_PLC_MS(),N);
clk := stime.0;
Q := clk XOR edge;
edge := CLK;

(* revision history
hm	16. dec 2007		rev 1.0
	original version

*)
END_FUNCTION_BLOCK

(* POU CLK_PRG, ST *)
	FUNCTION_BLOCK CLK_PRG
VAR_INPUT
	PT : TIME := t#10ms;
END_VAR
VAR_OUTPUT
	Q : BOOL := 0;
END_VAR
VAR
	init : BOOL := FALSE;
	last : TIME;
	tx: TIME;
END_VAR

(*
version 1.2	17 sep 2007
programmer 	hugo
tested by		tobias

clk_prg uses the internal sps time to generate a clock with programmable period time.
the period time is defined for 10ms .. 65s
the first cycle after start is a clk pulse and then depending on the programmed period time a delay.
every pulse is only valid for one cycle.
the accuracy of clk_prg is depending on the accuracy of the system clock.

*)
(* read system time *)
tx := DWORD_TO_TIME(T_PLC_MS());

(* initialize on startup *)
IF NOT init THEN
	init := TRUE;
	last := tx - pt;
END_IF;

(* generate output pulse when next_pulse is reached *)
IF tx - last >= pt THEN
	Q := TRUE;
	last := tx;
ELSE
	Q := FALSE;
END_IF;


(* revision hiostory

hm 25 feb 2007	rev 1.1
	rewritten code for higher performance
	pt can now be changed during runtime

hm	17. sep 2007	rev 1.2
	replaced time() with t_plc_ms() for compatibility reasons

*)
END_FUNCTION_BLOCK

(* POU CLK_PULSE, ST *)
FUNCTION_BLOCK CLK_PULSE
VAR_INPUT
	PT : TIME := t#10ms;
	N : INT := 0;
	rst : BOOL := 0;
END_VAR
VAR_OUTPUT
	Q : BOOL := 0;
	cnt : INT := 0;
	run : BOOL := 0;
END_VAR
VAR
	pti : TIME := t#0ms;
	next_pulse: TIME := T#0s;
	overflow: BOOL := FALSE;
	tx: TIME;
END_VAR

(*
version 1.1	17 sep 2007
programmer 	hugo
tested by		tobias

clk_pulse uses the internal sps time to generate a clock with programmable period time.
the period time is defined for 10ms .. 65s.
pulse generation is continuous if N = 0 and for n pulses otherwise.
if the period time is set to less then 10ms the min clock perid is 10ms.
the first cycle after start is a clk pulse and then depending on the programmed period time a delay.
every pulse is only valid for one cycle so that a edge trigger is not necessary
clk_prg depending on the accuracy of the system clock.

*)
(* read system *)
tx := DWORD_TO_TIME(T_PLC_MS());


IF rst THEN
	run := FALSE;
	pti := t#0ms;
	next_pulse := t#0ms;
	overflow := FALSE;
	Q := FALSE;
	cnt := 0;
ELSIF cnt <= N OR N = 0 THEN
	IF NOT run THEN
		next_pulse := tx;
		run := TRUE;
		IF pt < T#10ms THEN PTI := T#10ms; ELSE pti := pt; END_IF;
	END_IF;
	IF tx >= next_pulse AND NOT overflow AND (cnt < N OR N = 0) THEN
		Q := TRUE;
		cnt := cnt + 1;
		IF next_pulse + pti < next_pulse THEN
			overflow := TRUE;
		END_IF;
		next_pulse := next_pulse + pti;
	ELSE
		Q := FALSE;
		IF cnt = N THEN run := FALSE; END_IF
		IF tx <= next_pulse THEN overflow := FALSE; END_IF;
	END_IF;
END_IF

(* revision history
hm		4. aug 2006		rev 1.0
	original version

hm		17. sep 2007	rev 1.1
	replaced time() with T_PLC_S() fr compatblity reasons

*)
END_FUNCTION_BLOCK

(* POU CMP, ST *)
FUNCTION CMP : BOOL
VAR_INPUT
	X,Y : REAL;
	N : INT;
END_VAR
VAR
	tmp : REAL;
END_VAR


(*
	version 1.0	12 mar 2008
	programmer 	hugo
	tested by		tobias

this function checks two inputs x and y if they are identical with the first N digits
example : cmp(3.141516,3.141517,6 is true.

*)
tmp := ABS(x);
IF tmp > 0 THEN
	tmp :=	 EXP10(FLOOR(LOG(tmp))-N+1);
ELSE
	tmp := EXP10(tmp);
END_IF;
CMP := ABS(X - Y) < tmp;


(* revision history
hm		12. mar. 2008	rev 1.0
	original version

*)
END_FUNCTION

(* POU EXP10, ST *)
FUNCTION EXP10 : REAL
VAR_INPUT
	X : REAL;
END_VAR
VAR
END_VAR

(*
version 1.0	 2 dec 2007
programmer 	hugo
tested by		tobias

this function calculates the exponent to the basis 10
exp10(3) = 1000

*)
exp10 := EXP(X * 2.30258509299405);

(* revision history
hm	2. dec 2007		rev 1.0
	original version

*)
END_FUNCTION

(* POU FLOOR, ST *)
FUNCTION FLOOR : INT
VAR_INPUT
	X : REAL;
END_VAR
VAR
END_VAR


(*
version 1.1	21. mar. 2008
programmer 	hugo
tested by		tobias

This is a rounding function which returns the biggest possible integer which is less or equal to X.
floor(3.14) = 3
floor(-3.14) = -4

*)
FLOOR := REAL_TO_INT(X);
IF FLOOR > X THEN
	FLOOR := FLOOR - 1;
END_IF;

(* revision history
hm		7. feb 2007		rev 1.0
	originlal version

hm		21. mar. 2008	rev 1.1
	replaced trunc with real_to_int for compatibility reasons

*)
END_FUNCTION

(* POU CMUL, ST *)
FUNCTION CMUL : complex
VAR_INPUT
	X, Y : complex;
END_VAR
VAR
END_VAR

(*
version 1.0	21 feb 2008
programmer 	hugo
tested by	oscat

this function multiplies two complex numbers

*)
CMUL.re := X.re * Y.re - X.im * Y.im;
CMUL.im := X.re * Y.im + X.im * Y.re;

(* revision history
hm	21. feb 2008	rev 1.0
	original version

*)
END_FUNCTION

(* POU CONE_V, ST *)
FUNCTION CONE_V : REAL
VAR_INPUT
	rx : REAL;
	hx : REAL;
END_VAR
VAR
END_VAR

(*
version 1.1	4 dec 2007
programmer 	hugo
tested by		tobias

cone_V calculates the Volume of a cone

*)
cone_V := 1.047197551 * RX * RX * hx;

(* revision histroy
hm	17. oct 2007	rev 1.0
	original version

hm	4. dec 2007		rev 1.1
	changed code for better performance

hm	22. feb 2008	rev 1.2
	changed code for better performance
*)
END_FUNCTION

(* POU CONTROL_SET1, ST *)
FUNCTION_BLOCK CONTROL_SET1
VAR_INPUT
	Kt : REAL;
	Tt : REAL;
	PI : BOOL;
	PID : BOOL;
END_VAR
VAR_INPUT CONSTANT
	P_K : REAL := 0.5;
	PI_K : REAL := 0.45;
	PI_TN : REAL := 0.83;
	PID_K : REAL := 0.6;
	PID_TN : REAL := 0.5;
	PID_TV : REAL := 0.125;
END_VAR
VAR_OUTPUT
	KP : REAL;
	TN : REAL;
	TV : REAL;
	KI : REAL;
	KD : REAL;
END_VAR
VAR
END_VAR

(*
version 1.0	4 nov 2007
programmer 	hugo
tested by	tobias

takahashi calculates controller parameters for P, PI and PID controllers based on the ziegler nichols method.

*)
IF pi AND PID THEN
	KP := 0;
	TN := 0;
	TV := 0;
ELSIF PID THEN
	KP := PID_K * Kt;
	TN := PID_TN * Tt;
	TV := PID_TV * Tt;
ELSIF PI THEN
	KP := PI_K * Kt;
	TN := PI_TN * Tt;
ELSE
	KP := P_K * Kt;
END_IF;

(* KI and KD are calculated *)
IF tn > 0 THEN KI := KP / TN; ELSE KI := 0; END_IF;
KD := KP * TV;

(* revision history
hm	4. nov 2007		rev 1.0
	original version

*)
END_FUNCTION_BLOCK

(* POU CONTROL_SET2, ST *)
FUNCTION_BLOCK CONTROL_SET2
VAR_INPUT
	KS : REAL;
	TU : REAL;
	TG : REAL;
	PI : BOOL;
	PID : BOOL;
END_VAR
VAR_INPUT CONSTANT
	P_K : REAL := 1.0;
	PI_K : REAL := 0.9;
	PI_TN : REAL := 3.33;
	PID_K : REAL := 1.2;
	PID_TN : REAL := 2;
	PID_TV : REAL := 0.5;
END_VAR
VAR_OUTPUT
	KP : REAL;
	TN : REAL;
	TV : REAL;
	KI : REAL;
	KD : REAL;
END_VAR
VAR
	TX : REAL;
END_VAR

(*
version 1.0	4 nov 2007
programmer 	hugo
tested by	tobias

takahashi calculates controller parameters for P, PI and PID controllers based on the ziegler nichols method.

*)
IF TU > 0 AND KS > 0 THEN TX := TG/TU/KS; END_IF;
IF pi AND PID THEN
	KP := 0;
	TN := 0;
	TV := 0;
ELSIF PID THEN
	KP := PID_K * TX;
	TN := PID_TN * TU;
	TV := PID_TV * TU;
ELSIF PI THEN
	KP := PI_K * TX;
	TN := PI_TN * TU;
ELSE
	KP := P_K * TX;
END_IF;

(* KI and KD are calculated *)
IF TN > 0 THEN KI := KP / TN; ELSE KI := 0; END_IF;
KD := KP * TV;

(* revision history
hm	4. nov 2007		rev 1.0
	original version

*)
END_FUNCTION_BLOCK

(* POU COTH, ST *)
FUNCTION COTH : REAL
VAR_INPUT
	X : REAL;
END_VAR
VAR
END_VAR


(*
version 1.3	10. mar 2008
programmer 	hugo
tested by		tobias

this function calculates the cotangens hyperbolicus

*)
IF X > 20 THEN
	cotH :=1;
ELSIF X < -20 THEN
	COTH := -1;
ELSE
	COTH := 1 + 2 / (EXP(X * 2) - 1);
END_IF;


(* revision histroy
hm		12.1.2007	rev 1.0
	original version

hm		1.12.2007	rev 1.1
	changed code to improve performance

hm		8. jan 2008	rev 1.2
	further improvement in performance

hm		10. mar 2008	rev 1.3
	extended range of valid inputs to +/- INV
	changed formula for better accuracy
*)
END_FUNCTION

(* POU COUNT_BR, ST *)
FUNCTION_BLOCK COUNT_BR
VAR_INPUT
	SET : BOOL;
	IN : BYTE;
	UP : BOOL;
	DN : BOOL;
	STEP : BYTE := 1;
	MX : BYTE := 255;
	RST : BOOL;
END_VAR
VAR_OUTPUT
	CNT : BYTE;
END_VAR
VAR
	last_up: BOOL;
	last_dn: BOOL;
END_VAR

(*
	version 1.0	16 jan 2008
	programmer 	hugo
	tested BY	tobias

Count_BR is a byte counter with independen up and dn inputs. the counter counts from 0 to mx and continues at 0 after is has reached mx
a step input sets the counters stepping width.

*)
IF rst THEN
	cnt := 0;
ELSIF set THEN
	cnt := LIMIT(0,in,mx);
ELSIF up AND NOT last_up THEN
	cnt := INT_TO_BYTE(inc(cnt,step,mx));
ELSIF dn AND NOT last_dn THEN
	cnt := INT_TO_BYTE(inc(cnt,-step,mx));
END_IF;
last_up := up;
last_dn := dn;

(* revision history
hm	16. jan 2008	rev 1.0
	original version

*)
END_FUNCTION_BLOCK

(* POU INC, ST *)
FUNCTION INC : INT
VAR_INPUT
	X : INT;
	D : INT;
	M : INT;
END_VAR
VAR
END_VAR


(*
version 1.1	15. jan 2008
programmer 	hugo
tested by		tobias

This is a increment function which increments the input X by the value D and compares the result with M.
if the output exceeds M it will continue to count from 0 again.

*)
INC := (X + D + M + 1) MOD (M + 1);

(* revision history
hm	7. feb 2007		REV 1.0
	original version

hm	15. jan 2008	rev 1.1
	allow for neagtive increment

*)
END_FUNCTION

(* POU COUNT_CHAR, ST *)
FUNCTION COUNT_CHAR : INT
VAR_INPUT
	str : STRING(STRING_LENGTH);
	chr : BYTE;
END_VAR
VAR
	l: INT;
	pt : POINTER TO BYTE;
	pos: INT;
END_VAR


(*
version 1.1	29. mar. 2008
programmer 		kurt
tested by		hugo

COUNT_CHAR counts how often a character CHAR occurs within a string STR.

*)
PT := ADR(str);
l := LEN(str);
COUNT_CHAR := 0;
FOR pos := 1 TO l DO
	IF pt^ = CHR THEN COUNT_CHAR := COUNT_CHAR + 1; END_IF;
    PT := PT + 1;
END_FOR;


(* revision history
hm	29. feb 2008	rev 1.0
	original version

hm	29. mar. 2008	rev 1.1
	changed STRING to STRING(STRING_LENGTH)
*)
END_FUNCTION

(* POU COUNT_DR, ST *)
FUNCTION_BLOCK COUNT_DR
VAR_INPUT
	SET : BOOL;
	IN : DWORD;
	UP : BOOL;
	DN : BOOL;
	STEP : DWORD := 1;
	MX : DWORD := 255;
	RST : BOOL;
END_VAR
VAR_OUTPUT
	CNT : DWORD;
END_VAR
VAR
	last_up: BOOL;
	last_dn: BOOL;
END_VAR

(*
	version 1.0	12 jun 2008
	programmer 	hugo
	tested BY	tobias

Count_DR is a DWORD counter with independen up and dn inputs. the counter counts from 0 to mx and continues at 0 after is has reached mx
a step input sets the counters stepping width.

*)
IF rst THEN
	cnt := 0;
ELSIF set THEN
	cnt := LIMIT(0,in,mx);
ELSIF up AND NOT last_up THEN
	IF STEP > MX - CNT THEN
		CNT := CNT - MX + STEP - 1;
	ELSE
		CNT := CNT + STEP;
	END_IF
ELSIF dn AND NOT last_dn THEN
	IF STEP > CNT THEN
		CNT := CNT - STEP + MX + 1;
	ELSE
		CNT := CNT - STEP;
	END_IF;
END_IF;
last_up := up;
last_dn := dn;

(* revision history
hm	12. jun 2008	rev 1.0
	original version

*)
END_FUNCTION_BLOCK

(* POU CPOL, ST *)
FUNCTION CPOL : complex
VAR_INPUT
	L : REAL;
	A : REAL;
END_VAR
VAR
END_VAR

(*
version 1.0	21 feb 2008
programmer 	hugo
tested by	oscat

this function creates a complex numbers for the polar form with the inputs L (length) an A for Angle.

*)
CPOL.re := L * COS(A);
CPOL.im := L * SIN(A);


(* revision history
hm	21. feb 2008	rev 1.0
	original version

*)
END_FUNCTION

(* POU CPOW, ST *)
FUNCTION CPOW : complex
VAR_INPUT
	X : complex;
	Y : Complex;
END_VAR
VAR
END_VAR

(*
version 1.0	21 feb 2008
programmer 	hugo
tested by	oscat

this function calculates the complex power function x to the power of y

*)
CPOW := CEXP(CMUL(Y,CLOG(X)));


(* revision history
hm	21. feb 2008	rev 1.0
	original version

*)
END_FUNCTION

(* POU CRC_CHECK, ST *)
FUNCTION CRC_CHECK : BOOL
VAR_INPUT
	pt : POINTER TO ARRAY[0..32000] OF BYTE;
	size : UINT;
END_VAR
VAR_INPUT CONSTANT
	Polynom_L : DWORD;
	Polynom_32 : BOOL;
END_VAR
VAR
END_VAR

(*
version 1.1	16. mar. 2008
programmer 	hugo
tested by		tobias

CRC_CHECK checks a block of data for a crc checksum and returns true is the checksum is 0 and therfore a error free data transmission.
the CRC Polynom is specified with the config variable Polynom_L which holds the lowest 32 bits of the polynom and Polynom_33 which holds bit 33 of the Polynom.
A Polynom x4 + X + 1 is represented by 10011.
The input data is an array of byte of any size, the function is called by CRC_CHECK(ADR(array),SIZEOF(array)).

*)
CRC_CHECK := CRC_GEN(pt, size, polynom_L, polynom_32, 0, 0, FALSE, FALSE) = 0;


(* typical crc polynoms

CRC-4-ITU 			x4 + x + 1 					(ITU G.704, p. 12) 	0x3 or 0xC (0x9)
CRC-5-ITU 			x5 + x4 + x2 + 1 			(ITU G.704, p. 9) 	0x15 or 0x15 (0x0B)
CRC-5-USB 			x5 + x2 + 1 				(use: USB token packets) 	0x05 or 0x14 (0x9)
CRC-6-ITU 			x6 + x + 1 					(ITU G.704, p. 3) 	0x03 or 0x30 (0x21)
CRC-7 				x7 + x3 + 1 				(use: telecom systems, MMC) 	0x09 or 0x48 (0x11)
CRC-8-ATM 			x8 + x2 + x + 1 				(use: ATM HEC) 	0x07 or 0xE0 (0xC1)
CRC-8-CCITT 		x8 + x7 + x3 + x2 + 1 		(use: 1-Wire bus) 	0x8D or 0xB1 (0x63)
CRC-8-Dallas/Maxim 	x8 + x5 + x4 + 1 			(use: 1-Wire bus) 	0x31 or 0x8C (0x19)
CRC-8 				x8 + x7 + x6 + x4 + x2 + 1 	0xD5 or 0xAB (0x57)
CRC-8-SAE J1850 	x8 + x4 + x3 + x2 + 1 		0x1D or 0xB8
CRC-10 				x10 + x9 + x5 + x4 + x + 1 	0x233 or 0x331 (0x263)
CRC-12 				x12 + x11 + x3 + x2 + x + 1 (use: telecom systems) 	0x80F or 0xF01 (0xE03)
CRC-15-CAN 			x15 + x14 + x10 + x8 + x7 + x4 + x3 + 1 	0x4599 or 0x4CD1 (0x19A3)
CRC-16-Fletcher 	Not a CRC; see Fletcher's checksum 	Used in Adler-32 A & B CRCs
CRC-16-CCITT 	x16 + x12 + x5 + 1 (XMODEM,X.25, V.41, Bluetooth, PPP, IrDA; known as "CRC-CCITT") 	0x1021 or 0x8408 (0x0811)
CRC-16-IBM 	x16 + x15 + x2 + 1 (USB, many others; also known as "CRC-16") 	0x8005 or 0xA001 (0x4003)
CRC-24-Radix-64 	x24 + x23 + x18 + x17 + x14 + x11 + x10 + x7 + x6 + x5 + x4 + x3 + x + 1 	0x864CFB or 0xDF3261 (0xBE64C3)
CRC-32-Adler 	Not a CRC; see Adler-32 	See Adler-32
CRC-32-MPEG2 	x32 + x26 + x23 + x22 + x16 + x12 + x11 + x10 + x8 + x7 + x5 + x4 + x2 + x + 1 	0x04C11DB7 or 0xEDB88320 (0xDB710641) Also used in IEEE 802.3
CRC-32-IEEE 802.3 	x32 + x26 + x23 + x22 + x16 + x12 + x11 + x10 + x8 + x7 + x5 + x4 + x2 + x + 1 (V.42) 	0x04C11DB7 or 0xEDB88320 (0xDB710641)
CRC-32C (Castagnoli) 	x32 + x28 + x27 + x26 + x25 + x23 + x22 + x20 + x19 + x18 + x14 + x13 + x11 + x10 + x9 + x8 + x6 + 1 	0x1EDC6F41 or 0x82F63B78 (0x05EC76F1)
CRC-64-ISO 	x64 + x4 + x3 + x + 1 (use: ISO 3309) 	0x000000000000001B or 0xD800000000000000 (0xB000000000000001)
CRC-64-ECMA-182 	x64 + x62 + x57 + x55 + x54 + x53 + x52 + x47 + x46 + x45 + x40 + x39 + x38 + x37 + x35 + x33 + x32 + x31 + x29 + x27 + x24 + x23 + x22 + x21 + x19 + x17 + x13 + x12 + x10 + x9 + x7 + x4 + x + 1
(as described in ECMA-182 p.63) 	0x42F0E1EBA9EA3693 or 0xC96C5795D7870F42 (0x92D8AF2BAF0E1E85)

*)

(* revision history

hm		9.6.2007		rev 1.0		
	original version 

hm		16. mar. 2008	rev 1.1
	changed type of input size to uint
	improved code for better performance	
*)
END_FUNCTION

(* POU CRC_GEN, ST *)
FUNCTION CRC_GEN : DWORD

VAR_INPUT
	pt : POINTER TO ARRAY[0..32000] OF BYTE;
	size : UINT;
END_VAR
VAR_INPUT CONSTANT
	Polynom_L : DWORD;
	Polynom_32 : BOOL;
	init: DWORD := 0;
	XOR_out : DWORD;
	rev_in : BOOL;
	rev_out : BOOL;
END_VAR
VAR
	polynom : DWORD;
	p_length : INT;
	BS : BYTE;
	data : DWORD;
	count : BYTE;
	temp : BOOL;
	step: INT;
	s4: INT;
END_VAR

(*
version 1.4	16. mar. 2008
programmer 	hugo
tested by		tobias

CRC_GEN generates a CRC checksum from a block of data and returns  the checksum in a DWORD to be connected to the data for transmission.
the CRC Polynom is specified with the config variable Polynom_L which holds the lowest 32 bits of the polynom and Polynom_33 which holds bit 33 of the Polynom.
A Polynom x4 + X + 1 is represented by 10011.
The input data is an array of byte of any size, the function is called by CRC_GEN(ADR(array),SIZEOF(array)).

*)
(* check for polynom length and calculate p_length polynom will be aligned to high side of word*)
polynom := polynom_L;
IF polynom_32 THEN
	p_length := 33;
ELSE;
	p_length := 32;
	WHILE p_length > 0 AND NOT polynom.31 DO
		p_length := p_length - 1;
		Polynom := SHL(polynom,1);
	END_WHILE;
	Polynom := SHL(polynom,1);
END_IF;


(* load start code and first data byte for crc calculation *)
data := init;
IF rev_in THEN bs := reverse(pt^[0]); ELSE bs := pt^[0]; END_IF;

(* calcualte checksum *)
s4 := UINT_TO_INT(size) + 4;
WHILE step < s4 DO
	temp := data.31;
	data := SHL(data,1);
	data.0 := BS.7;
	bs := SHL(bs,1);
	count := count + 1;
	IF count = 8 THEN
		step := step + 1;
		count := 0;
		IF step < UINT_TO_INT(size) THEN
			IF rev_in THEN bs := reverse(pt^[step]); ELSE bs := pt^[step]; END_IF;
		END_IF;
	END_IF;
	(* check highest bit if true then xor polynom *)
	IF temp THEN data := data XOR polynom; END_IF;
END_WHILE;

(* reverse crc if necessary *)
IF rev_out THEN
	CRC_GEN.31 := data.31;
	FOR step := p_length TO 3 BY -1 DO
		data := SHL(data,1);
		CRC_GEN := SHR(CRC_GEN,1);
		CRC_GEN.31 := data.31;
	END_FOR;
ELSE
	CRC_GEN := data;
END_IF;

(* final XOR and align crc checksum to right side of dword *)
CRC_GEN := CRC_GEN XOR SHL(xor_out, 33 - p_length);
CRC_GEN := SHR(CRC_GEN,33 - p_length);


(* old code prior to rev 1.2
B1 := pt^[0];
IF size > 1 THEN B2 := pt^[1]; ELSE B2 := 0; END_IF;
IF size > 2 THEN B3 := pt^[2]; ELSE B3 := 0; END_IF;
IF size > 3 THEN B4 := pt^[3]; ELSE B4 := 0; END_IF;
IF size > 4 THEN BS := pt^[4]; ELSE BS := 0; END_IF;
data := DWord_of_Byte(B4,B3,B2,B1);

WHILE step < size DO
	temp := data.31;
	data := SHL(data,1);
	data.0 := BS.7;
	bs := SHL(bs,1);
	count := count + 1;
	IF count = 8 THEN
		step := step + 1;
		count := 0;
		IF step + 4 < size THEN bs := pt^[step+ 4]; END_IF;
	END_IF;
	(* check highest bit if true then xor polynom *)
	IF temp = TRUE THEN
		data := data XOR polynom;
	END_IF;
END_WHILE;

(* align crc checksum to right side of dword *)
CRC_GEN := SHR(data,32 - p_length +1);
*)


(* typical crc polynoms

CRC-4-ITU 			x4 + x + 1 					(ITU G.704, p. 12) 	0x3 or 0xC (0x9)
CRC-5-ITU 			x5 + x4 + x2 + 1 			(ITU G.704, p. 9) 	0x15 or 0x15 (0x0B) Bluetooth
CRC-5-USB 			x5 + x2 + 1 				(use: USB token packets) 	0x05 or 0x14 (0x9)
CRC-6-ITU 			x6 + x + 1 					(ITU G.704, p. 3) 	0x03 or 0x30 (0x21)
CRC-7 				x7 + x3 + 1 				(use: telecom systems, MMC) 	0x09 or 0x48 (0x11)
CRC-8-ATM 			x8 + x2 + x + 1 				(use: ATM HEC) 	0x07 or 0xE0 (0xC1)
CRC-8-CCITT 		x8 + x7 + x3 + x2 + 1 		(use: 1-Wire bus) 	0x8D or 0xB1 (0x63)
CRC-8-Dallas/Maxim 	x8 + x5 + x4 + 1 			(use: 1-Wire bus) 	0x31 or 0x8C (0x19)
CRC-8 				x8 + x7 + x6 + x4 + x2 + 1 	0xD5 or 0xAB (0x57)
CRC-8-SAE J1850 	x8 + x4 + x3 + x2 + 1 		0x1D or 0xB8
CRC-10 				x10 + x9 + x5 + x4 + x + 1 	0x233 or 0x331 (0x263)
CRC-12 				x12 + x11 + x3 + x2 + x + 1 (use: telecom systems) 	0x80F or 0xF01 (0xE03)
CRC-15-CAN 			x15 + x14 + x10 + x8 + x7 + x4 + x3 + 1 	0x4599 or 0x4CD1 (0x19A3)
CRC-16-Fletcher 	Not a CRC; see Fletcher's checksum 	Used in Adler-32 A & B CRCs
CRC-16-CCITT 	x16 + x12 + x5 + 1 (XMODEM,X.25, V.41, Bluetooth, PPP, IrDA; known as "CRC-CCITT") 	0x1021 or 0x8408 (0x0811)
CRC-16-IBM 	x16 + x15 + x2 + 1 (USB, many others; also known as "CRC-16") 	0x8005 or 0xA001 (0x4003)
CRC-24-Radix-64 	x24 + x23 + x18 + x17 + x14 + x11 + x10 + x7 + x6 + x5 + x4 + x3 + x + 1 	0x864CFB or 0xDF3261 (0xBE64C3)
CRC-32-Adler 	Not a CRC; see Adler-32 	See Adler-32
CRC-32-MPEG2 	x32 + x26 + x23 + x22 + x16 + x12 + x11 + x10 + x8 + x7 + x5 + x4 + x2 + x + 1 	0x04C11DB7 or 0xEDB88320 (0xDB710641) Also used in IEEE 802.3
CRC-32-IEEE 802.3 	x32 + x26 + x23 + x22 + x16 + x12 + x11 + x10 + x8 + x7 + x5 + x4 + x2 + x + 1 (V.42) 	0x04C11DB7 or 0xEDB88320 (0xDB710641)
CRC-32C (Castagnoli) 	x32 + x28 + x27 + x26 + x25 + x23 + x22 + x20 + x19 + x18 + x14 + x13 + x11 + x10 + x9 + x8 + x6 + 1 	0x1EDC6F41 or 0x82F63B78 (0x05EC76F1)
CRC-64-ISO 	x64 + x4 + x3 + x + 1 (use: ISO 3309) 	0x000000000000001B or 0xD800000000000000 (0xB000000000000001)
CRC-64-ECMA-182 	x64 + x62 + x57 + x55 + x54 + x53 + x52 + x47 + x46 + x45 + x40 + x39 + x38 + x37 + x35 + x33 + x32 + x31 + x29 + x27 + x24 + x23 + x22 + x21 + x19 + x17 + x13 + x12 + x10 + x9 + x7 + x4 + x + 1
(as described in ECMA-182 p.63) 	0x42F0E1EBA9EA3693 or 0xC96C5795D7870F42 (0x92D8AF2BAF0E1E85)

*)

(* revision history

hm		9.6.2007		rev 1.0		
	original version 

hm		11.9.2007		rev 1.1
	deleted unused variable i

hm		9. oct 2007 	rev 1.2
	added init code for crc and xor_out
	added refelct in and reflect_out (rev_in und Rev_out)

hm		2. jan 2008		rev 1.3
	small changes for performance improvements

hm		16. mar. 2008	rev 1.4
	changed type of input size to uint
*)
END_FUNCTION

(* POU REVERSE, ST *)
FUNCTION REVERSE : BYTE
VAR_INPUT
	IN : BYTE;
END_VAR
VAR
END_VAR

(*
	version 1.1	18. feb 2008
	programmer 	hugo
	tested BY		tobias

This function reverses the bits of a byte so that after execution bit 7 is at bit 0 location and so forth.

*)
reverse := SHL(in,7) OR SHR(in,7) OR (ROR(in,3) AND 2#01000100) OR (ROL(in,3) AND 2#00100010)
	OR (SHL(in,1) AND 2#00010000) OR (SHR(in,1) AND 2#00001000);


(* revision history
hm		9.oct 2007		rev 1.0
	original version

hm		18. feb 2008	rev 1.1
	improved performance
*)
END_FUNCTION

(* POU CSIN, ST *)
FUNCTION CSIN : complex
VAR_INPUT
	X : complex;
END_VAR
VAR
END_VAR

(*
version 1.0	21 feb 2008
programmer 	hugo
tested by	oscat

this function calculates the sinus function of a complex number

*)
CSIN.re := cosH(X.im) * SIN(X.re);
CSIN.im := sinH(X.im) * COS(X.re);


(* revision history
hm	21. feb 2008	rev 1.0
	original version

*)
END_FUNCTION

(* POU CSINH, ST *)
FUNCTION CSINH : complex
VAR_INPUT
	X : complex;
END_VAR
VAR
END_VAR

(*
version 1.0	21 feb 2008
programmer 	hugo
tested by	oscat

this function calculates the sinus function of a complex number

*)
CSINH.re := sinH(X.re) * COS(X.im);
CSINH.im := cosH(X.re) * SIN(X.im);


(* revision history
hm	21. feb 2008	rev 1.0
	original version

*)
END_FUNCTION

(* POU CSUB, ST *)
FUNCTION CSUB : complex
VAR_INPUT
	X, Y : complex;
END_VAR
VAR
END_VAR

(*
version 1.0	21 feb 2008
programmer 	hugo
tested by	oscat

this function subtracts two complex numbers

*)
CSUB.re := X.re - Y.re;
CSUB.im := X.im - Y.im;

(* revision history
hm	21. feb 2008	rev 1.0
	original version

*)
END_FUNCTION

(* POU CTAN, ST *)
FUNCTION CTAN : complex
VAR_INPUT
	X : complex;
END_VAR
VAR
	temp : REAL;
END_VAR

(*
version 1.0	21 feb 2008
programmer 	hugo
tested by	oscat

this function calculates the tangens function of a complex number

*)
temp := 1 / (COS(2 * x.re) + cosH( 2 * x.im));
CTAN.re := temp * SIN(2 * x.re);
CTAN.im := temp * sinH(2 * x.im);


(* revision history
hm	21. feb 2008	rev 1.0
	original version

*)
END_FUNCTION

(* POU CTANH, ST *)
FUNCTION CTANH : complex
VAR_INPUT
	X : complex;
END_VAR
VAR
	temp : REAL;
END_VAR

(*
version 1.0	21 feb 2008
programmer 	hugo
tested by	oscat

this function calculates the complex hyperbolictangens

*)
temp := 1 /(cosH(2 * x.re) + COS(2 * x.im));
CTANH.re := temp * sinH(2 * x.re);
CTANH.im := temp * SIN(2 * x.im);


(* revision history
hm	21. feb 2008	rev 1.0
	original version

*)
END_FUNCTION

(* POU CTRL_IN, ST *)
FUNCTION CTRL_IN : REAL
VAR_INPUT
	SET_POINT, ACTUAL, NOISE : REAL;
END_VAR


(*
version 1.0	2. jun 2008
programmer 	hugo
tested by		tobias


*)
(* calculate the process error DIFF *)
CTRL_IN := DEAD_ZONE(SET_POINT - ACTUAL, NOISE);


(* revision history
hm 	2. jun. 2008 	rev 1.0
	original version

*)
END_FUNCTION

(* POU DEAD_ZONE, ST *)
FUNCTION DEAD_ZONE : REAL
VAR_INPUT
	X : REAL;
	L : REAL;
END_VAR
VAR
END_VAR

(*
version 1.1	14 jun. 2008
programmer 	hugo
tested by	oscat

dead_zone2 is a linear transfer function which follows a linear function except for x is close to 0.
Y = X if abs(x) > L otherwise its 0.

*)
IF ABS(x) > L THEN
	dead_zone := X;
ELSE
	dead_zone := 0;
END_IF;

(* revision history
hm	12. feb. 2007	rev 1.0
	original version

hm	14. jun. 2008	rev 1.1
	improved performance

*)
END_FUNCTION

(* POU CTRL_OUT, ST *)
FUNCTION_BLOCK CTRL_OUT
VAR_INPUT
	CI, OFFSET, MAN_IN, LIM_L, LIM_H : REAL;
	MANUAL : BOOL;
END_VAR
VAR_OUTPUT
	Y : REAL;
	LIM : BOOL;
END_VAR


(*
version 1.0	2. jun 2008
programmer 	hugo
tested by		tobias


*)
IF manual THEN
	Y := MAN_IN + OFFSET;
ELSE
	Y := CI + OFFSET;
END_IF;


(* Limit the output *)
IF Y >= LIM_H THEN
	Y := LIM_H;
	LIM := TRUE;
ELSIF Y <= lim_L THEN
	Y := LIM_L;
	LIM := TRUE;
ELSE
	LIM := FALSE;
END_IF;



(* revision history
hm 	2. jun. 2008 	rev 1.0
	original version

*)
END_FUNCTION_BLOCK

(* POU CTRL_PI, ST *)
FUNCTION_BLOCK CTRL_PI
VAR_INPUT
	ACT, SET, SUP, OFS, M_I : REAL;
	MAN : BOOL;
	RST : BOOL := FALSE;
	KP : REAL := 1.0;
	KI : REAL := 1.0;
	LL : REAL := -1000;
	LH : REAL := 1000;
END_VAR
VAR_OUTPUT
	Y : REAL;
	DIFF : REAL;
	LIM : BOOL;
END_VAR
VAR
	pi : FT_PIWL;
	co : CTRL_OUT;
END_VAR

(*
version 2.0	30. jun 2008
programmer 	hugo
tested by	oscat

FT_PI is a PI controller with manual functionality.
The PID controller works according to the fomula Y = e *(KP+ KI * INTEG(e) ) + offset, while e = set_point - actual.
a rst will reset all internal data, while a switch to manual will cause the controller to follow the function Y = manual_in + offset.
limit_h and Limit_l set the possible output range of Y.
the output flags lim will signal that the output limits are active and overflow will signal that the integrator has reached its limits.

since rev 1.1 the "trapezregel is used for more accuracy.
rev 1.2 added selective integratin which means the integrative component is only active within a small range of the target value 
this avoids the integrator to go to limits while an input setpoint change happened and is only causing overshoots.
the int_band is by default 100 which means the int is active all the time and if set to for example to 0.1 the integrator is only active
while the input is between 0.9 and 1.1 of the set_point value.

default values for KP = 1, TN = 1, TV = 1, LIMIT_L = -1000, LIMIT_H = +1000.
*)
DIFF := CTRL_IN(SET, ACT, SUP);
pi(in := DIFF, kp := KP, ki := KI, lim_l := LL, lim_h := LH, rst := RST);
co(ci := pi.Y, OFFSET := OFS, man_in := M_I, lim_l := LL, lim_h := LH, manual := MAN);
Y := co.Y;
LIM := co.LIM;


(* revision history
hm 	31.10.2007 		rev 1.0
	original version

hm	3.11.2007		rev 1.1
	added noise input to filter noise
	added output diff
	set limit output false when output is within limits
	overfolw was not set correctly

hm	5. jan 2008		rev 1.2
	improved performance

hm	20. jun. 2008	rev 2.0
	rewritten using new modular approach

*)
END_FUNCTION_BLOCK

(* POU FT_PIWL, ST *)
FUNCTION_BLOCK FT_PIWL
VAR_INPUT
	IN : REAL;
	KP : REAL := 1.0;
	KI : REAL := 1.0;
	LIM_L : REAL := -1E38;
	LIM_H : REAL := 1E38;
	RST : BOOL := FALSE;
END_VAR
VAR_OUTPUT
	Y : REAL;
	LIM : BOOL;
END_VAR
VAR
	init: BOOL;
	tx: DWORD;
	tc : REAL;
	t_last: DWORD;
	in_last : REAL;
	i: REAL;
	p: REAL;
END_VAR

(*
version 1.0	13. jun 2008
programmer 	hugo
tested by	tobias

FT_PIWL is a PI controller.
The PID controller works according to the fomula Y = IN *(KP+ KI * INTEG(e) ).
a rst will reset the integrator to 0
lim_h and Lim_l set the possible output range of the controller.
the output flag lim will signal that the output limits are active.
the integrator ist equipped with anti wind-up circuitry which limits trhe total output ranke to lim_l and lim_h

default values for KP = 1, KI = 1, ILIM_L = -1E37, iLIM_H = +1E38.
*)
(* initialize at power_up *)
IF NOT init OR RST THEN
	init := TRUE;
	in_last := in;
	t_last := T_PLC_US();
	i := 0;
	tc := 0;
ELSE
	(* read last cycle time in Microseconds *)
	tx := T_PLC_US();
	tc := DWORD_TO_REAL(tx - t_last);
	t_last := tx;

	(* calculate proportional part *)
	p := KP * IN;

	(* run integrator *)
	i := (IN + in_last) * 5E-7 * KI * tc + i;
	in_last := IN;

	(* calculate output Y *)
	Y := p + i;

	(* check output for limits *)
	IF Y >= LIM_H THEN
		Y := LIM_H;
		i := LIM_H - p;
		LIM := TRUE;
	ELSIF Y <= LIM_L THEN
		Y := LIM_L;
		i := LIM_L - p;
		LIM := TRUE;
	ELSE
		LIM := FALSE;
	END_IF;
END_IF;




(* revision history
hm 	13. jun. 2008 	rev 1.0
	original version

*)
END_FUNCTION_BLOCK

(* POU CTRL_PID, ST *)
FUNCTION_BLOCK CTRL_PID
VAR_INPUT
	ACT, SET, SUP, OFS, M_I : REAL;
	MAN : BOOL;
	RST : BOOL := FALSE;
	KP : REAL := 1.0;
	TN : REAL := 1.0;
	TV : REAL := 1.0;
	LL : REAL := -1000;
	LH : REAL := 1000;
END_VAR
VAR_OUTPUT
	Y : REAL;
	DIFF : REAL;
	LIM : BOOL;
END_VAR
VAR
	pid : FT_PIDWL;
	co : CTRL_OUT;
END_VAR



(*
version 2.0	30. jun. 2008
programmer 	hugo
tested by	oscat

FT_PI is a PI controller with manual functionality.
The PID controller works according to the fomula Y = e *(KP+ KI * INTEG(e) ) + offset, while e = set_point - actual.
a rst will reset all internal data, while a switch to manual will cause the controller to follow the function Y = manual_in + offset.
limit_h and Limit_l set the possible output range of Y.
the output flags lim will signal that the output limits are active.

*)
DIFF := CTRL_IN(SET, ACT, SUP);
pid(in := DIFF, kp := KP, tn := TN, tv := TV, lim_l := LL, lim_h := LH, rst := RST);
co(ci := pid.Y, OFFSET := OFS, man_in := M_I, lim_l := LL, lim_h := LH, manual := MAN);
Y := co.Y;
LIM := co.LIM;



(* revision history

hm 1.12.2006	 	rev 1.1
	changed algorithm to trapezregel for higher accuracy.

hm 3.1.2007		rev 1.2
	added integ_band to select when the integrator is active.

hm	3.3.2007		rev 1.3
	added default values to inputs KP, TN, TV, LIMIT_L und LIMIT_H.

hm 31.oct 2007	rev 1.4
	total rewrite of the module to avoid failures when one of the limits is 0

hm	3.11.2007	rev 1.5
	added noise input to filter noise
	added output diff
	set limit output false when output is within limits
	overfolw was not set correctly

hm	5. jan 2008	rev 1.6
	improved code for better performance
*)
END_FUNCTION_BLOCK

(* POU FT_PIDWL, ST *)
FUNCTION_BLOCK FT_PIDWL
VAR_INPUT
	IN : REAL;
	KP : REAL := 1.0;
	TN : REAL := 1.0;
	TV : REAL := 1.0;
	LIM_L : REAL := -1E38;
	LIM_H : REAL := 1E38;
	RST : BOOL := FALSE;
END_VAR
VAR_OUTPUT
	Y : REAL;
	LIM : BOOL;
END_VAR
VAR
	piwl : FT_PIWL;
	diff : FT_DERIV;
END_VAR

(*
version 1.0	13. jun 2008
programmer 	hugo
tested by		tobias

FT_PIDW is a PID controller with dynamic wind_up reset.
The PID controller works according to the fomula Y = KP *(IN + KI * INTEG(e) + DERIV(e) ).
a rst will reset the integrator to 0
lim_h and Lim_l set the possible output range of the internal integrator.
the output flags lim will signal that the output limits are active.

default values for KP = 1, KI = 1, ILIM_L = -1E37, iLIM_H = +1E38.
*)
(* if rst then *)
IF rst THEN
	piwl(rst := TRUE);
	piwl.RST := FALSE;
ELSE
	(* run PIWL controller first *)
	(* we need to check if TN = 0 and do alternative calls *)
	IF TN = 0 THEN
		piwl(in := IN, KP := KP, KI := 0, LIM_L := LIM_L, LIM_H := LIM_H);
	ELSE
		piwl(in := IN, KP := KP, KI := 1/TN, LIM_L := LIM_L, LIM_H := LIM_H);
	END_IF;

	(* run differentiator and add_to_output *)
	diff(IN := IN, K := TV);
	Y := piwl.Y + diff.out;

	(* limit the output *)
	IF Y < LIM_L THEN
		LIM := TRUE;
		Y := LIM_L;
	ELSIF Y > LIM_H THEN
		LIM := TRUE;
		Y := LIM_H;
	ELSE
		LIM := FALSE;
	END_IF;
END_IF;



(* revision history
hm 	13. jun. 2008 	rev 1.0
	original version


*)
END_FUNCTION_BLOCK

(* POU FT_DERIV, ST *)
FUNCTION_BLOCK FT_DERIV
VAR_INPUT
	in : REAL;
	K : REAL := 1;
	run : BOOL := 1;
END_VAR
VAR_OUTPUT
	out : REAL;
END_VAR
VAR
	old: REAL;
	tx: DWORD;
	last: DWORD;
	init: BOOL;
END_VAR


(*
version 1.3	29 oct 2007
programmer 	hugo
tested by		tobias

FT_deriv calculates the derivate over the signal "in" with Faktor "K".
a run input enables or stops the calculation, if left unconnected its true and therfore the calculation is executed.
if K is not specified the default is 1.

*)
(* read system time *)
tx := T_PLC_US();

(* init on firsat startup *)
IF NOT init THEN
	init := TRUE;
	old := in;
	last := tx;
END_IF;
IF run AND tx - last > 0 THEN
	out := (in - old) / DWORD_TO_REAL(tx - last) * 1000000.0 * K;
	last := tx;
ELSE
	out := 0;
	last := tx;
END_IF;
old := in;


(*
hm 3.1.2007			rev 1.1
	added init code for startup
	set the default for K to 1

hm	15. sep 2007	rev 1.2
	replaced Time() with T_PLC_US for compatibility and performance reasons
	increased accuracy and work in microseconds internally

hm 29 oct 2007	rev 1.3
	prohibit calculation when tx - last = 0 to avoid division by 0 and increase accuracy on fast systems
*)
END_FUNCTION_BLOCK

(* POU CTRL_PWM, ST *)
FUNCTION_BLOCK CTRL_PWM
VAR_INPUT
	CI, MAN_IN : REAL;
	MANUAL : BOOL;
	F : REAL;
END_VAR
VAR_OUTPUT
	Q : BOOL;
END_VAR
VAR
	PW : PWM_DC;
END_VAR

(*
version 1.0	3. jun 2008
programmer 	hugo
tested by		tobias


*)
IF MANUAL THEN
	PW(F := F, DC := MAN_IN);
ELSE
	PW(F := F, DC := CI);
END_IF;
Q := PW.Q;



(* revision history
hm 	3. jun. 2008 	rev 1.0
	original version

*)
END_FUNCTION_BLOCK

(* POU PWM_DC, ST *)
FUNCTION_BLOCK PWM_DC
VAR_INPUT
	F : REAL;
	DC : REAL;
END_VAR
VAR_OUTPUT
	Q : BOOL;
END_VAR
VAR
	clk: CLK_Prg;
	pulse: TP_R;
END_VAR

(*
	version 1.2	27 nov 2007
	programmer 	oscat
	tested BY		oscat

this signal generator generates a square wave signal which is specified by the frequency and the duty cycle
*)
IF F > 0 THEN
	CLK(PT := REAL_TO_TIME(1000/F));
	Pulse(in := clk.Q, pt := REAL_TO_TIME(1000/F*DC));
	Q := pulse.Q;
END_IF;

(* revision history

hm		25. feb 2007	rev 1.1
	recoded in st for better performance and better portability

hm		27. nov 2007	rev 1.2
	avoid divide by 0 when F = 0
*)
END_FUNCTION_BLOCK

(* POU TP_R, ST *)
FUNCTION_BLOCK TP_R
VAR_INPUT
	in : BOOL;
	PT : TIME;
END_VAR
VAR_OUTPUT
	Q : BOOL := 0;
	ET : TIME := t#0ms;
END_VAR
VAR
	edge : BOOL := FALSE;
	start : TIME := t#0ms;
	tx: TIME;
END_VAR

(*
version 1.1	17 sep 2007
programmer 	hugo
tested by		tobias

retriggerable edge triggered pulse similar to TP but with a retrigger function
if the pt input is 0 then output is always low.
*)
(* read system_time *)
tx := DWORD_TO_TIME(T_PLC_MS());

(* rising edge trigger *)
IF in AND NOT edge THEN
	start := Tx;
	IF pt > t#0ms THEN Q := TRUE; END_IF;
END_IF;
edge := in;
IF q THEN
	et := Tx - start;
	IF et >= PT THEN
		Q := FALSE;
		et := t#0ms;
	END_IF;
END_IF;


(* revision history
hm	4. aug 2006		rev 1.0
	original version

hm	17. sep 2007	rev 1.1
	replaced time() with T_PLC_MS() for compatibility reasons
	
*)
END_FUNCTION_BLOCK

(* POU D_TRIG, ST *)
FUNCTION_BLOCK D_TRIG
VAR_INPUT
	in : DWORD;
END_VAR
VAR_OUTPUT
	Q : BOOL;
	X : DWORD;
END_VAR
VAR
	last_in : DWORD;
END_VAR

(*
version 1.1	19. feb 2008
programmer 	hugo
tested by		tobias

this block is similar to the IEC Standard R_trig and F_trig but it monitors a DWORD, WORD or Byte Variable instead and generated an Output Pulse for one cycle only when the input has changed.
an additional output x (Dword) will state the chage of the input.
Example: the input has chaged from 0001 to 0010 then the output x will be 2.

*)
Q := in <> last_in;
X := in - last_in;
last_in := in;


(* revision history

hm 	4.09.2007		rev 1.0
	original version released

hm	19. feb. 2008	rev 1.1
	performance improvement
*)
END_FUNCTION_BLOCK

(* POU DATE_ADD, ST *)
FUNCTION DATE_ADD : DATE
VAR_INPUT
	idate : DATE;
	D : INT;
	W : INT;
	M : INT;
	Y : INT;
END_VAR
VAR
	mo: INT;
	yr : INT;
END_VAR


(*
version 1.3	22. mar 2008
programmer 	hugo
tested by		tobias

date_add adds days, weeks, month or years to a date.
negative inputs are allowed for subtraction.

*)
DATE_ADD := DWORD_TO_DATE(DATE_TO_DWORD(idate) + 86400 * INT_TO_DWORD(d) + 604800 * INT_TO_DWORD(w));
mo := month(date_add);
yr := year(date_add) + y + FLOOR(INT_TO_REAL(mo + m - 1) / 12.0);
mo := mo + (ABS(m) MOD 12) * SGN(m);
IF mo < 1 THEN
	mo := mo + 12;
ELSIF mo > 12 THEN
	mo := mo - 12;
END_IF;
date_add := set_Date(yr,mo,day_of_month(date_add));



(* revision history

hm 27.12.2006		rev 1.0

hm 12.4.2007		rev 1.1
	corrected an error while date would be incorrect when year  = 0

hm	1.11.2007		rev 1.2
	added int_to_dword stetements to avoid possible overrun with möller ecp4

hm	22. mar. 2008	rev 1.3
	fixed some bugs when month was negative
*)
END_FUNCTION

(* POU MONTH, ST *)
FUNCTION MONTH : INT
VAR_INPUT
	idate : DATE;
END_VAR
VAR
END_VAR

(*
version 1.1	1 okt 2007
programmer 	hugo
tested by	tobias

returns the month of a year

*)
month := day_of_year(idate);
IF leap_of_Date(idate) THEN
	CASE month OF
		1..31 	:	month := 1;
		32..60	:	month := 2;
		61..91	:	month := 3;
		92..121 :	month := 4;
		122..152:	month := 5;
		153..182:	month := 6;
		183..213:	month := 7;
		214..244:	month := 8;
		245..274:	month := 9;
		275..305:	month := 10;
		306..335:	month := 11;
		336..366:	month := 12;
	END_CASE;
ELSE
	CASE month OF
		1..31 	:	month := 1;
		32..59	:	month := 2;
		60..90	:	month := 3;
		91..120 :	month := 4;
		121..151:	month := 5;
		152..181:	month := 6;
		182..212:	month := 7;
		213..243:	month := 8;
		244..273:	month := 9;
		274..304:	month := 10;
		305..334:	month := 11;
		335..365:	month := 12;
	END_CASE;
END_IF;


(* old code used in rev 1.0
month := STRING_TO_INT(MID(DATE_TO_STRING(idate),2,8));
*)

(* revision history
hm	1. aug 2006		rev 1.0
	original version	

hm	1. okt 2007		rev 1.1
	replaced old code (string conversion) with mathematics
	the execution time is now multiple times faster.

*)
END_FUNCTION

(* POU DAY_OF_YEAR, ST *)
FUNCTION DAY_OF_YEAR : INT
VAR_INPUT
	idate : DATE;
END_VAR
VAR
END_VAR

(*
version 1.2	4 jan 2008
programmer 	hugo
tested by		tobias

calculates the day of the year

*)
day_of_year := DWORD_TO_INT((DATE_TO_DWORD(idate) - DATE_TO_DWORD(year_begin(year(idate))))/86400) + 1;


(* version before rev 1.2
IF step7 THEN
	day_of_year := DWORD_TO_INT(DATE_TO_DWORD(idate)/86400 + 726483 - TRUNC((year(idate)-1)*365.25));
ELSE
	day_of_year := DWORD_TO_INT(DATE_TO_DWORD(idate)/86400 + 719178 - TRUNC((year(idate)-1)*365.25));
END_IF;
*)


(* revivision history
hm	4. aug 2007		rev 1.0
	original version

hm	1. okt 2007		rev 1.1
	added compatibility to STEP7

hm	4. jan 2008		rev 1.2
	changed code for better performance
*)
END_FUNCTION

(* POU YEAR_BEGIN, ST *)
FUNCTION YEAR_BEGIN : DATE
VAR_INPUT
	y : INT;
END_VAR
VAR
END_VAR

(*
version 1.2	7. Apr. 2008
programmer 	hugo
tested by	tobias

returs the date of january 1st for the given year  
the function works for dates from 1970 - 2099 

*)
year_begin := DWORD_TO_DATE(SHR(INT_TO_DWORD(y) * 1461 - 2878169,2)*86400);



(* revision history
hm	19. dec 2007	rev 1.0
	original version

hm	4. jan 2008		rev 1.1
	formula for step7 was incorrect during leap years

hm	7. apr. 2008	rev 1.2
	deleted unused step7 code
*)
END_FUNCTION

(* POU YEAR, ST *)
FUNCTION YEAR : INT
VAR_INPUT
	idate : DATE;
END_VAR
VAR
END_VAR

(*
version 1.3	7. apr. 2008
programmer 	hugo
tested by		tobias

returs the year of a date  
the function works for dates from 1970 - 2099 

*)
year := DWORD_TO_INT((DATE_TO_DWORD(idate)+43200) / 31557600 + 1970);


(* code used prior to rev 1.1
year := DWORD_TO_INT((DATE_TO_DWORD(idate)/864+71954300)/36525);
*)

(* revision history
hm	4. aug 2006		rev 1.0
	original version

hm	1. okt 2007		rev 1.1
	corrected error in algorithm
	adjustment for S7 compatibility

hm	23.12.2007		rev 1.2
	changed code for better performance

hm	7. apr. 2008	rev 1.3
	deleted unused step7 code
*)
END_FUNCTION

(* POU LEAP_OF_DATE, ST *)
FUNCTION LEAP_OF_DATE : BOOL
VAR_INPUT
	idate : DATE;
END_VAR
VAR
END_VAR

(*
version 1.2	8 jan 2008
programmer 	hugo
tested by		tobias

leap_year is true if the tested year is a leap year  

*)
leap_of_Date := SHL(DWORD_TO_INT((DATE_TO_DWORD(idate)+43200) / 31557600)+2,14) = 0;


(* change history

2.10.2006		rev 1.1
the function now calls leap_year to accomodate further accuracy.
the function now works for any year from 1970 to 2100

8. jan 2008		rev 1.2
	improved code for better performance
*)
END_FUNCTION

(* POU SET_DATE, ST *)
FUNCTION SET_DATE : DATE
VAR_INPUT
	year : INT;
	month : INT;
	day : INT;
END_VAR
VAR
	count : DWORD;
END_VAR

(*
version 1.6	7. apr. 2008
programmer 	hugo
tested by	tobias

creates a date output from year, month and day of month   

*)
count := SHR(INT_TO_DWORD(year) * 1461 - 2878173,2)+INT_TO_DWORD(day);

IF month < 5 THEN
	IF month < 3 THEN
		IF month = 2 THEN count := count + 31; END_IF;
	ELSE
		IF month = 4 THEN
			IF SHL(year,14) = 0 THEN count := count + 91; ELSE count := count + 90; END_IF;
		ELSE (* month = 3 *)
			IF SHL(year,14) = 0 THEN count := count + 60; ELSE count := count + 59; END_IF;
		END_IF;
	END_IF;
ELSIF month < 9 THEN
	IF month < 7 THEN
		IF month = 6 THEN
			IF SHL(year,14) = 0 THEN count := count + 152; ELSE count := count + 151; END_IF;
		ELSE (* month = 5 *)
			IF SHL(year,14) = 0 THEN count := count + 121; ELSE count := count + 120; END_IF;
		END_IF;
	ELSE
		IF month = 8 THEN
			IF SHL(year,14) = 0 THEN count := count + 213; ELSE count := count + 212; END_IF;
		ELSE (* month = 7 *)
			IF SHL(year,14) = 0 THEN count := count + 182; ELSE count := count + 181; END_IF;
		END_IF;
	END_IF;
ELSE (* month is 9 or higher *)
	IF month < 11 THEN
		IF month = 10 THEN
			IF SHL(year,14) = 0 THEN count := count + 274; ELSE count := count + 273; END_IF;
		ELSE (* month = 9 *)
			IF SHL(year,14) = 0 THEN count := count + 244; ELSE count := count + 243; END_IF;
		END_IF;
	ELSE
		IF month = 12 THEN
			IF SHL(year,14) = 0 THEN count := count + 335; ELSE count := count + 334; END_IF;
		ELSE (* month = 11 *)
			IF SHL(year,14) = 0 THEN count := count + 305; ELSE count := count + 304; END_IF;
		END_IF;
	END_IF;
END_IF;
set_Date := DWORD_TO_DATE(count * 86400);

(*  code before rev 1.4
leap := leap_year(year);
IF STEP7 THEN
	count := SHR((year-1)*1461-2905932+day*4,2);
ELSE
	count := SHR((year-1)*1461-2876712+day*4,2);
END_IF;
CASE month OF
2:	count := count + 31;
3:	IF leap THEN count := count + 60; ELSE count := count + 59; END_IF;
4:	IF leap THEN count := count + 91; ELSE count := count + 90; END_IF;
5:	IF leap THEN count := count + 121; ELSE count := count + 120; END_IF;
6:	IF leap THEN count := count + 152; ELSE count := count + 151; END_IF;
7:	IF leap THEN count := count + 182; ELSE count := count + 181; END_IF;
8:	IF leap THEN count := count + 213; ELSE count := count + 212; END_IF;
9:	IF leap THEN count := count + 244; ELSE count := count + 243; END_IF;
10:	IF leap THEN count := count + 274; ELSE count := count + 273; END_IF;
11:	IF leap THEN count := count + 305; ELSE count := count + 304; END_IF;
12:	IF leap THEN count := count + 335; ELSE count := count + 334; END_IF;
END_CASE;
set_Date := DWORD_TO_DATE(count * 86400);
*)

(* old code before rev 1.3
leap := leap_year(year);
IF STEP7 THEN
	count := TRUNC((year-1)*365.25-726483+day);
ELSE
	count := TRUNC((year-1)*365.25-719178+day);
END_IF;
CASE month OF
2:	count := count + 31;
3:	IF leap THEN count := count + 60; ELSE count := count + 59; END_IF;
4:	IF leap THEN count := count + 91; ELSE count := count + 90; END_IF;
5:	IF leap THEN count := count + 121; ELSE count := count + 120; END_IF;
6:	IF leap THEN count := count + 152; ELSE count := count + 151; END_IF;
7:	IF leap THEN count := count + 182; ELSE count := count + 181; END_IF;
8:	IF leap THEN count := count + 213; ELSE count := count + 212; END_IF;
9:	IF leap THEN count := count + 244; ELSE count := count + 243; END_IF;
10:	IF leap THEN count := count + 274; ELSE count := count + 273; END_IF;
11:	IF leap THEN count := count + 305; ELSE count := count + 304; END_IF;
12:	IF leap THEN count := count + 335; ELSE count := count + 334; END_IF;
END_CASE;
set_Date := DWORD_TO_DATE(count * 86400);
*)




(* revision history
hm	4. aug. 2006	rev 1.0
	original version

hm	19 sep. 2007	rev 1.1
	use function leap_year to calculate leap year, more exceptions are handled

hm	1. okt	2007	rev 1.2
	added compatibility to step7

hm	16.dec 2007	rev 1.3
	changed code to improove performance

hm	3. jan. 2008	rev 1.4
	further improvements in performance

hm	16. mar. 2008	rev 1.5
	added type conversions to avoid warnings under codesys 3.0

hm	7. apr. 2008	rev 1.6
	deleted unused step7 code
*)
END_FUNCTION

(* POU DAY_OF_MONTH, ST *)
FUNCTION DAY_OF_MONTH : INT
VAR_INPUT
	idate : DATE;
END_VAR
VAR
END_VAR

(*
version 1.4	8. jan 2008
programmer 	hugo
tested by	tobias

returns the day OF month for any DATE

*)
day_of_month := day_of_year(idate);
IF leap_of_Date(idate) THEN
	CASE day_of_month OF
		32..60	:	day_of_month := day_of_month - 31;
		61..91	:	day_of_month := day_of_month - 60;
		92..121 :	day_of_month := day_of_month - 91;
		122..152:	day_of_month := day_of_month - 121;
		153..182:	day_of_month := day_of_month - 152;
		183..213:	day_of_month := day_of_month - 182;
		214..244:	day_of_month := day_of_month - 213;
		245..274:	day_of_month := day_of_month - 244;
		275..305:	day_of_month := day_of_month - 274;
		306..335:	day_of_month := day_of_month - 305;
		336..366:	day_of_month := day_of_month - 335;
	END_CASE;
ELSE
	CASE day_of_month OF
		32..59	:	day_of_month := day_of_month - 31;
		60..90	:	day_of_month := day_of_month - 59;
		91..120 :	day_of_month := day_of_month - 90;
		121..151:	day_of_month := day_of_month - 120;
		152..181:	day_of_month := day_of_month - 151;
		182..212:	day_of_month := day_of_month - 181;
		213..243:	day_of_month := day_of_month - 212;
		244..273:	day_of_month := day_of_month - 243;
		274..304:	day_of_month := day_of_month - 273;
		305..334:	day_of_month := day_of_month - 304;
		335..365:	day_of_month := day_of_month - 334;
	END_CASE;
END_IF;


(*
this function is simple but took too long with 133 us
the problem is date_to_string is far too slow
day_of_month := STRING_TO_INT(RIGHT(DATE_TO_STRING(idate),2));

Revision history

hm 22.1.2007		rev 1.1
	deleted unused variable day_in_year and day_in_year_begin

hm	1. okt 2007		rev 1.2
	changed code to use day_of_year and leap_of_date
	added compatibility to STEP7

hm	8. oct 2007		rev 1.3
	deleted unused variable yr

hm	8. jan 2008		rev 1.4
	improved performance
*)
END_FUNCTION

(* POU DAY_OF_DATE, ST *)
FUNCTION DAY_OF_DATE : DINT
VAR_INPUT
	idate : DATE;
END_VAR
VAR
END_VAR


(*
	version 1.3	7. apr. 2008
	programmer 	oscat
	tested BY	oscat

DAY_OF_DATE returns the days since 1.1.1970

*)
day_of_date := DWORD_TO_DINT(DATE_TO_DWORD(idate) / 86400);


(* revision history
hm		16.9.2007		rev 1.0
	original version

hm		1. okt 2007		rev 1.1
	added step7 compatibility

hm		22. mar. 2008	rev 1.2
	changed output from int to Dint because the total date range is 49710 days

hm		7. apr. 2008	rev 1.3
	deleted unused step7 code

*)
END_FUNCTION

(* POU DAY_TO_TIME, ST *)
FUNCTION DAY_TO_TIME : TIME
VAR_INPUT
	input : REAL;
END_VAR
VAR
END_VAR

(*
version 1.0	4 aug 2006
programmer 	hugo
tested by		tobias

converts an amount of days in real to time 
*)
day_to_time := DWORD_TO_TIME(REAL_TO_DWORD(input * 86400000));
END_FUNCTION

(* POU DAYS_DELTA, ST *)
FUNCTION DAYS_DELTA : DINT
VAR_INPUT
	date_1 : DATE;
	date_2 : DATE;
END_VAR
VAR
END_VAR

(*
version 1.2	22. mar. 2008
programmer 	hugo
tested by		tobias

days_delta calculates the days between two dates. the days are calculated date_2 - date_1.

*)
days_delta := day_of_date(date_2) - day_of_date(date_1);

(* revision history
hm	27. dec 2006	rev 1.0
	original version

hm	16.9.2007		rev 1.1
	coorected an error in formula and changed algorithm to show positive and negative delta

hm	22. mar. 2008	rev 1.2
	changed output from int to dint because the total date range is 49710 days
*)
END_FUNCTION

(* POU DCF77, ST *)
FUNCTION_BLOCK DCF77
VAR_INPUT
	REC : BOOL;
	SET : BOOL;
	SDT : DT;
	DSI : BOOL;
END_VAR
VAR_INPUT CONSTANT
	SYNC_TIMEOUT : TIME := t#2m;
	TIME_OFFSET : INT := 1;
	DST_EN : BOOL := TRUE;
END_VAR
VAR_OUTPUT
	TP : BOOL;
	DS : BOOL;
	WDAY : INT;
	ERROR : BOOL := TRUE;
	RTC : DT;
	RTC1 : DT;
	MSEC : INT;
	SYNC : BOOL;
END_VAR
VAR
	mez : DT;
	utc : DT;
	state : INT;
	edge: BOOL;
	tx : TIME;
	ty: TIME;
	last : TIME;
	bits : ARRAY[0..58] OF BOOL;
	cnt : INT;
	i : INT;
	old_time : DT;
	minute : INT;
	hour : INT;
	day : INT;
	month : INT;
	year : INT;
	last_sync: TIME;
	t1: TIME;
	tz: TIME;
	init: BOOL;
END_VAR


(*
version 1.9	19. apr. 2008
programmer 	hugo
tested by		tobias

this is a decoder for a DCF77 signal.
the decoder decodes the DCF77 signal and checks for a valid Date_Time.
since the dcf77 signal is only secured with a simple parity the decoder waits for two consecutive valid transmissions before it sets the output signals.
given a valid reception by the receiver the decoder can take up to 3 minutes to start its clocks the first time.
after a valid signal is detected the error output goes low and dignals a valid dcf signal from the receiver.
a tp is only valid for one program cycle to allow for external rtc setting.
after a valid signal is detected two independent internal clocks are started (RTC and RTC1), the seconds  of these clocks are generated by software since the dcf signal is only valid for minutes.
rtc is always utc ( world time) and rtc1 can be set to any time zone by setting the time_zone_offset and enabling dst for automatic summertime.
a sync output signals the the rtc and rtc1 are in sync with the dcf77 signal, if the dcf77 signal is lost for more then the sync time the sync output goes low
but the rtc and rtc1 outputs keep running based on software timing until a valid dcf77 signal is received again and triggers the clock.
in addition a millisecond output gives further resolutionof the clocks.
a dst output shows if daylight saving time is enables and the weekday output shows which day of week currently is ( 1= monday ... 7= sunday).

*)
(* if tp was set it should only be active for 1 cycle *)
TP := FALSE;

(* read system time *)
t1 := DWORD_TO_TIME(T_PLC_MS());
tx := t1 - last;

IF rec XOR edge THEN
	edge := rec;
	IF NOT rec AND tx > t#1700ms AND tx < t#2000ms THEN
		(* start condition reached *)
		state := 0;
		tp := NOT error;
	ELSIF NOT rec AND tx > t#700ms AND tx < t#1000ms THEN
		(* second switch detected *)
		IF state < 58 THEN state := state +1; ELSE state := 0; END_IF;
	ELSIF rec AND tx  < t#120ms THEN
		(* bit 0 detected  *)
		bits[state] := 0;
	ELSIF rec AND tx > t#120ms AND tx < t#250ms THEN
		(* bit 1 detected *)
		bits[state] := 1;
	ELSE
		(* error condition received signal is not valid *)
		error := TRUE;
		state := 0;
	END_IF;
	last := last + tx;
	IF rec AND state = 58 THEN
		error := FALSE;

		(* decode the bits and check for possible errors *)
		IF bits[0] OR NOT (bits[17] XOR bits[18]) OR NOT bits[20] THEN error := TRUE; END_IF;
		(* decode minute *)
		MINUTE := 0;
		MINUTE.0 := bits[21];
		MINUTE.1 := bits[22];
		MINUTE.2 := bits[23];
		MINUTE.3 := bits[24];
		IF bits[25] THEN MINUTE := MINUTE + 10; END_IF;
		IF bits[26] THEN MINUTE := MINUTE + 20; END_IF;
		IF bits[27] THEN MINUTE := MINUTE + 40; END_IF;
		IF MINUTE > 59 OR (bits[21] XOR bits[22] XOR bits[23] XOR bits[24] XOR bits[25] XOR bits[26] XOR bits[27] XOR bits[28]) THEN error := TRUE; END_IF;

		(* decode hour *)
		HOUR := 0;
		HOUR.0 := bits[29];
		HOUR.1 := bits[30];
		HOUR.2 := bits[31];
		HOUR.3 := bits[32];
		IF bits[33] THEN HOUR := HOUR + 10; END_IF;
		IF bits[34] THEN HOUR := HOUR +20; END_IF;
		IF HOUR > 23 OR (bits[29] XOR bits[30] XOR bits[31] XOR bits[32] XOR bits[33] XOR bits[34] XOR bits[35]) THEN error := TRUE; END_IF;

		(* decode day of month *)
		day := 0;
		day.0 := bits[36];
		day.1 := bits[37];
		day.2 := bits[38];
		day.3 := bits[39];
		IF bits[40] THEN day := day + 10; END_IF;
		IF bits[41] THEN day := day + 20; END_IF;
		IF day > 31 THEN error := TRUE; END_IF;

		(* decode day of week *)
		wday := 0;
		wday.0 := bits[42];
		wday.1 := bits[43];
		wday.2 := bits[44];
		IF wday > 7 OR wday < 1 THEN error := TRUE; END_IF;

		(* decode month *)
		MONTH := 0;
		MONTH.0 := bits[45];
		MONTH.1 := bits[46];
		MONTH.2 := bits[47];
		MONTH.3 := bits[48];
		IF bits[49] THEN MONTH := MONTH +10; END_IF;
		IF MONTH > 12 THEN error := TRUE; END_IF;

		(* decode year *)
		YEAR := 0;
		YEAR.0 := bits[50];
		YEAR.1 := bits[51];
		YEAR.2 := bits[52];
		YEAR.3 := bits[53];
		IF bits[54] THEN YEAR := YEAR + 10; END_IF;
		IF bits[55] THEN YEAR := YEAR + 20; END_IF;
		IF bits[56] THEN YEAR := YEAR + 40; END_IF;
		IF bits[57] THEN YEAR := YEAR + 80; END_IF;

		(* check parity for bits 36 to 58 *)
		cnt := 0;
		FOR i := 36 TO 58 DO IF bits[i] THEN cnt := cnt + 1; END_IF; END_FOR;
		IF NOT EVEN(cnt) THEN error := TRUE; END_IF;

		(* time must be valid for two cycles to clear error flag *)
		IF NOT error THEN
			(* set outputs *)
			old_time := mez;
			IF YEAR >= 70 THEN YEAR := YEAR + 1900; ELSE YEAR := YEAR + 2000; END_IF;
			mez := SET_DT(YEAR,MONTH,day,HOUR,MINUTE,0);
			DS := bits[17];
			IF DS THEN
				UTC := DWORD_TO_DT(DT_TO_DWORD(mez) - 7200);
			ELSE
				UTC := DWORD_TO_DT(DT_TO_DWORD(mez) - 3600);
			END_IF

			(* set trigger signal only if the receiver has received 2 successive minutes *)
			IF mez <> old_time + t#1m THEN error := TRUE ; END_IF;
		END_IF;
	END_IF;
END_IF;

(* this portion implements a free running clock which is triggered by the dcf77 signal *)
tz := DWORD_TO_TIME(INT_TO_DWORD(ABS(time_offset))* 3600000);

(* input sdt is copied to utc at first power up *)
IF NOT init OR SET THEN
	init := TRUE;
	utc := sdt;
	tp := TRUE;
	DS := DSI;
END_IF;

